// ---- Library/10_Machine/18_HMI_Handshake/DUTs/IOMonitor/ST_Wheelhouse_Layer.TcDUT
TYPE ST_Wheelhouse_Layer :
STRUCT
	Line : ARRAY[1..20] OF BOOL;
END_STRUCT
END_TYPE

// ---- Library/10_Machine/18_HMI_Handshake/DUTs/IOMonitor/UNI_HMI_WheelHouseInput.TcDUT
TYPE UNI_HMI_WheelHouseInput :
UNION
	arWheelHouseInput : ARRAY[1..400] OF BOOL;
	List :ST_WheelhouseInput;
END_UNION
END_TYPE

// ---- Library/10_Machine/18_HMI_Handshake/DUTs/IOMonitor/UNI_HMI_WheelHouseInput2.TcDUT
TYPE UNI_HMI_WheelHouseInput2 :
UNION
	arWheelHouseInput : ARRAY[1..400] OF BOOL;
	List :ST_WheelhouseInput;
END_UNION
END_TYPE

// ---- Library/10_Machine/18_HMI_Handshake/DUTs/Shipping/ST_Auto_Shipping.TcDUT
TYPE
    ST_Auto_Shipping :
    STRUCT
    END_STRUCT
END_TYPE

// ---- Library/10_Machine/18_HMI_Handshake/DUTs/Shipping/ST_HalfAuto_Shipping.TcDUT
TYPE
    ST_HalfAuto_Shipping :
    STRUCT
    END_STRUCT
END_TYPE

// ---- Library/10_Machine/18_HMI_Handshake/DUTs/Shipping/ST_HMI_ShippingArea.TcDUT
TYPE
    ST_HMI_ShippingArea :
    STRUCT
        //提供新的馬達
    END_STRUCT
END_TYPE

// ---- Library/10_Machine/18_HMI_Handshake/DUTs/Shipping/ST_Manual_Shipping.TcDUT
TYPE
    ST_Manual_Shipping :
    STRUCT
		FanucRobot : ST_Manual_FanucRobot;
    END_STRUCT
END_TYPE

// ---- Library/10_Machine/18_HMI_Handshake/DUTs/Status/ST_AllocateStatus.TcDUT
TYPE
    ST_AllocateStatus :
    STRUCT
    END_STRUCT
END_TYPE

// ---- Library/10_Machine/18_HMI_Handshake/DUTs/Status/ST_Auto_Status.TcDUT
TYPE ST_Auto_Status :
STRUCT
END_STRUCT
END_TYPE

// ---- Library/10_Machine/18_HMI_Handshake/DUTs/Status/ST_AXES_STATUS.TcDUT
TYPE ST_AXES_STATUS :
    STRUCT
        TurnTable       : ST_SINGLEAXIS_STATUS; 		// 圓盤 狀態
        Allocate        : ST_SINGLEAXIS_STATUS; 		// 圓帶 狀態
        Needle_X        : ST_SINGLEAXIS_STATUS; 		// 配針 X 狀態
        Needle_Y        : ST_SINGLEAXIS_STATUS; 		// 配針 Y 狀態
        OutRobot_X      : ST_SINGLEAXIS_STATUS; 		// 出料手臂 X 狀態
        OutRobot_Y      : ST_SINGLEAXIS_STATUS; 		// 出料手臂 Y 狀態
		RackMotor 		: ST_SINGLEAXIS_STATUS; 		// 補貨料架馬達 狀態
		ElvaterAxis		: ST_SINGLEAXIS_STATUS;			// 電梯 狀態
		HookAxis		: ST_SINGLEAXIS_STATUS;			// 勾盤 狀態
		FinishAxis		: ST_SINGLEAXIS_STATUS;			// 出料層架 狀態
    END_STRUCT
END_TYPE

// ---- Library/10_Machine/18_HMI_Handshake/DUTs/Status/ST_MotorStatus.TcDUT
TYPE
    ST_MotorStatus :
    STRUCT
        WareHouseCV_10          : ST_MotorMonitor;
        WareHouseCV_09          : ST_MotorMonitor;
        WareHouseCV_08          : ST_MotorMonitor;
        WareHouseCV_07          : ST_MotorMonitor;
        WareHouseCV_06          : ST_MotorMonitor;
        WareHouseCV_05          : ST_MotorMonitor;
        WareHouseCV_04          : ST_MotorMonitor;
        WareHouseCV_03          : ST_MotorMonitor;
        WareHouseCV_02          : ST_MotorMonitor;
        WareHouseCV_01          : ST_MotorMonitor;
        WareHouseCV_20          : ST_MotorMonitor;
        WareHouseCV_19          : ST_MotorMonitor;
        WareHouseCV_18          : ST_MotorMonitor;
        WareHouseCV_17          : ST_MotorMonitor;
        WareHouseCV_16          : ST_MotorMonitor;
        WareHouseCV_15          : ST_MotorMonitor;
        WareHouseCV_14          : ST_MotorMonitor;
        WareHouseCV_13          : ST_MotorMonitor;
        WareHouseCV_12          : ST_MotorMonitor;
        WareHouseCV_11          : ST_MotorMonitor;
        UpCV                    : ST_MotorMonitor;
        LowCV                   : ST_MotorMonitor;
        PullOutCV_A             : ST_MotorMonitor;
        PullOutCV_B             : ST_MotorMonitor;
        TransmitSameSideCV      : ST_MotorMonitor;
        TransmitDifferentSideCV : ST_MotorMonitor;
    END_STRUCT
END_TYPE

// ---- Library/10_Machine/18_HMI_Handshake/DUTs/Status/ST_SINGLEAXIS_STATUS.TcDUT
TYPE ST_SINGLEAXIS_STATUS :
    STRUCT
        ActPos    : LREAL; // Axis actual position with gear ratio
        ActVel    : LREAL; // Axis actual velocity with gear ratio
        MotorTemp : LREAL; // Motor current tempture, if motor doesn't have temp sensor, this value will be zero.
        DriveTemp : LREAL; // Driver current tempture
        Homed     : BOOL; // Axis has homed 
        Error     : BOOL; // Axis has error
        CmdDone   : BOOL; // Axis Cmd completed
    END_STRUCT
END_TYPE

// ---- Library/10_Machine/18_HMI_Handshake/DUTs/Status/ST_CylinderStatus.TcDUT
TYPE
    ST_CylinderStatus :
    STRUCT
        UpCV_FeedInPress1             : ST_CylinderMonitor;
        UpCV_FeedInPress2             : ST_CylinderMonitor;
        UpCV_DiameterPress            : ST_CylinderMonitor;
        UpCV_CamaraPress1             : ST_CylinderMonitor;
        UpCV_CamaraPress2             : ST_CylinderMonitor;
        UpCV_CamaraPress3             : ST_CylinderMonitor;
        UpCV_CamaraPress4             : ST_CylinderMonitor;
        UpCV_Block1                   : ST_CylinderMonitor;
        UpCV_Block2                   : ST_CylinderMonitor;
        UpCV_Block3                   : ST_CylinderMonitor;
        UpCV_DiameterHoriz            : ST_CylinderMonitor;
        UpCV_DiameterVert             : ST_CylinderMonitor;
        UpCV_DiameterClamp            : ST_CylinderMonitor;
        StackPush                     : ST_CylinderMonitor;
        PullOutCV_AsidePress1         : ST_CylinderMonitor;
        PullOutCV_AsidePress2         : ST_CylinderMonitor;
        PullOutCV_AsideBlock          : ST_CylinderMonitor;
        PullOutCV_BsidePress1         : ST_CylinderMonitor;
        PullOutCV_BsidePress2         : ST_CylinderMonitor;
        PullOutCV_BsideBlock          : ST_CylinderMonitor;
        LowCV_Press1                  : ST_CylinderMonitor;
        LowCV_Press2                  : ST_CylinderMonitor;
        LowCV_Press3                  : ST_CylinderMonitor;
        LowCV_Press4                  : ST_CylinderMonitor;
        LowCV_Block1                  : ST_CylinderMonitor;
        LowCV_Block2                  : ST_CylinderMonitor;
        AllocateRobot_LeftVert1       : ST_CylinderMonitor;
        AllocateRobot_LeftVert2       : ST_CylinderMonitor;
        AllocateRobot_RightVert1      : ST_CylinderMonitor;
        AllocateRobot_RightVert2      : ST_CylinderMonitor;
        AllocateRobot_LeftClamp1      : ST_CylinderMonitor;
        AllocateRobot_LeftClamp2      : ST_CylinderMonitor;
        AllocateRobot_RightClamp1     : ST_CylinderMonitor;
        AllocateRobot_RightClamp2     : ST_CylinderMonitor;
        RoundBelt_WorkZone_Press      : ST_CylinderMonitor;
        RoundBelt_WorkZone_Plug       : ST_CylinderMonitor;
        RoundBelt_ChargeZone_Plug     : ST_CylinderMonitor;
        RoundBelt_TransmitCVZone_Plug : ST_CylinderMonitor;
        OutRobot_AsideVert            : ST_CylinderMonitor;
        OutRobot_BsideVert            : ST_CylinderMonitor;
        OutRobot_AsideClamp           : ST_CylinderMonitor;
        OutRobot_BsideClamp           : ST_CylinderMonitor;
        TransmitCV_CamaraHoriz        : ST_CylinderMonitor;
        DifferentSizeCV_Press2        : ST_CylinderMonitor;
        DifferentSizeCV_Press1        : ST_CylinderMonitor;
        DifferentSizeCV_Block1        : ST_CylinderMonitor;
        SameSizeCV_Press4             : ST_CylinderMonitor;
        SameSizeCV_Press3             : ST_CylinderMonitor;
        SameSizeCV_Press2             : ST_CylinderMonitor;
        SameSizeCV_Press1             : ST_CylinderMonitor;
        SameSizeCV_Block2             : ST_CylinderMonitor;
        SameSizeCV_Block1             : ST_CylinderMonitor;
        Turntable_Press               : ST_CylinderMonitor;
    END_STRUCT
END_TYPE

// ---- Library/10_Machine/18_HMI_Handshake/DUTs/Status/ST_HalfAuto_Status.TcDUT
TYPE ST_HalfAuto_Status :
STRUCT
END_STRUCT
END_TYPE

// ---- Library/10_Machine/18_HMI_Handshake/DUTs/Status/ST_HMI_MachineStatus.TcDUT
TYPE
    ST_HMI_MachineStatus :
    STRUCT
        Axes      : ST_AXES_STATUS;	  //馬達狀態
        Cylinders : ST_CylinderStatus;//汽缸狀態
        Motor     : ST_MotorStatus;	  //軌道狀態
    END_STRUCT
END_TYPE

// ---- Library/10_Machine/18_HMI_Handshake/DUTs/Status/ST_Manual_Status.TcDUT
TYPE ST_Manual_Status :
STRUCT
	Cylinders : ST_CylinderStatus;
END_STRUCT
END_TYPE

// ---- Library/10_Machine/18_HMI_Handshake/DUTs/Status/ST_ShippingStatus.TcDUT
TYPE ST_ShippingStatus :
STRUCT
END_STRUCT
END_TYPE

// ---- Library/10_Machine/18_HMI_Handshake/DUTs/Status/ST_StorageStatus.TcDUT
TYPE ST_StorageStatus :
STRUCT
END_STRUCT
END_TYPE

// ---- Library/10_Machine/18_HMI_Handshake/DUTs/Storage/ST_Auto_Storage.TcDUT
TYPE
    ST_Auto_Storage :
    STRUCT
    END_STRUCT
END_TYPE

// ---- Library/10_Machine/18_HMI_Handshake/DUTs/Storage/ST_HalfAuto_Storage.TcDUT
TYPE
    ST_HalfAuto_Storage :
    STRUCT
    END_STRUCT
END_TYPE

// ---- Library/10_Machine/18_HMI_Handshake/DUTs/Storage/ST_HMI_ControlConvery.TcDUT
TYPE
    ST_HMI_ControlConvery :
    STRUCT
		//A倉軌道
        WareHouseCV_10  : ST_MotorCommand;
        WareHouseCV_09  : ST_MotorCommand;
        WareHouseCV_08  : ST_MotorCommand;
        WareHouseCV_07  : ST_MotorCommand;
        WareHouseCV_06  : ST_MotorCommand;
        WareHouseCV_05  : ST_MotorCommand;
        WareHouseCV_04  : ST_MotorCommand;
        WareHouseCV_03  : ST_MotorCommand;
        WareHouseCV_02  : ST_MotorCommand;
        WareHouseCV_01  : ST_MotorCommand;
		//B倉軌道
        WareHouseCV_20  : ST_MotorCommand;
        WareHouseCV_19  : ST_MotorCommand;
        WareHouseCV_18  : ST_MotorCommand;
        WareHouseCV_17  : ST_MotorCommand;
        WareHouseCV_16  : ST_MotorCommand;
        WareHouseCV_15  : ST_MotorCommand;
        WareHouseCV_14  : ST_MotorCommand;
        WareHouseCV_13  : ST_MotorCommand;
        WareHouseCV_12  : ST_MotorCommand;
        WareHouseCV_11  : ST_MotorCommand;
		
        UpCV            : ST_Manual_UpCV;			//上層入料軌道
        LowCV        	: ST_Manual_LowCV;			//下層出料軌道
		PullOutCV       : ST_Manual_PullOutCV;      // 空盒以及拔針軌道
        TransCV         : ST_Manual_TransCV;        // 同尺寸以及配針軌道
    END_STRUCT
END_TYPE

// ---- Library/10_Machine/18_HMI_Handshake/DUTs/Storage/ST_Manual_FanucRobot.TcDUT
TYPE ST_Manual_FanucRobot :
STRUCT
	ClampA_Open  		: BOOL; // True: set clampA open 
	ClampA_Close 		: BOOL; // True: Set ClampA Close
	ClampB_Open  		: BOOL; // True: Set ClampB Open
	ClampB_Close 		: BOOL; // True: Set ClampB Close
	ByPassClampSensor   : BOOL; // True : Bypass clampA and clampB
END_STRUCT
END_TYPE

// ---- Library/10_Machine/18_HMI_Handshake/DUTs/Storage/ST_Manual_Rack.TcDUT
TYPE ST_Manual_Rack :
STRUCT
	Axis                : ST_Manual_Axis; // RoundBelt Axis controll
END_STRUCT
END_TYPE

// ---- Library/10_Machine/18_HMI_Handshake/DUTs/Storage/ST_Manual_UpCV.TcDUT
TYPE
    ST_Manual_UpCV :
    STRUCT
        FeedInPress1  : ST_SignleValve;
        FeedInPress2  : ST_SignleValve;
        DiameterPress : ST_SignleValve;
        CamaraPress1  : ST_SignleValve;
        CamaraPress2  : ST_SignleValve;
        CamaraPress3  : ST_SignleValve;
        CamaraPress4  : ST_SignleValve;
        Block1        : ST_SignleValve;
        Block2        : ST_SignleValve;
        Block3        : ST_SignleValve;
        DiameterHoriz : ST_SignleValve;
        DiameterVert  : ST_SignleValve;
        DiameterClamp : ST_SignleValve;
        StackPush     : ST_SignleValve;
		CameraBlow	  : BOOL;
        UpCV          : ST_MotorCommand;
    END_STRUCT
END_TYPE

// ---- Library/10_Machine/18_HMI_Handshake/DUTs/Storage/ST_Manual_LowCV.TcDUT
TYPE
    ST_Manual_LowCV :
    STRUCT
        Press1 : ST_SignleValve;
        Press2 : ST_SignleValve;
        Press3 : ST_SignleValve;
        Press4 : ST_SignleValve;
        Block1 : ST_SignleValve;
        Block2 : ST_SignleValve;
        LowCV  : ST_MotorCommand;
    END_STRUCT
END_TYPE

// ---- Library/10_Machine/18_HMI_Handshake/DUTs/Storage/ST_Manual_Storage.TcDUT
TYPE
    ST_Manual_Storage :
    STRUCT
        WareHouseCV_10 : ST_MotorCommand;
        WareHouseCV_09 : ST_MotorCommand;
        WareHouseCV_08 : ST_MotorCommand;
        WareHouseCV_07 : ST_MotorCommand;
        WareHouseCV_06 : ST_MotorCommand;
        WareHouseCV_05 : ST_MotorCommand;
        WareHouseCV_04 : ST_MotorCommand;
        WareHouseCV_03 : ST_MotorCommand;
        WareHouseCV_02 : ST_MotorCommand;
        WareHouseCV_01 : ST_MotorCommand;
        WareHouseCV_20 : ST_MotorCommand;
        WareHouseCV_19 : ST_MotorCommand;
        WareHouseCV_18 : ST_MotorCommand;
        WareHouseCV_17 : ST_MotorCommand;
        WareHouseCV_16 : ST_MotorCommand;
        WareHouseCV_15 : ST_MotorCommand;
        WareHouseCV_14 : ST_MotorCommand;
        WareHouseCV_13 : ST_MotorCommand;
        WareHouseCV_12 : ST_MotorCommand;
        WareHouseCV_11 : ST_MotorCommand;
        UpCV           : ST_Manual_UpCV;
        LowCV          : ST_Manual_LowCV;
		FanucRobot : ST_Manual_FanucRobot;
		RackMotor :ST_Manual_Rack;
    END_STRUCT
END_TYPE

// ---- Library/10_Machine/18_HMI_Handshake/OLD_DUTs/DataCore/E_BoxHookPoint.TcDUT
{attribute 'qualified_only'}
{attribute 'strict'}
TYPE E_BoxHookPoint :
(
	
	Origin 		:= 0,
	Station_1	:= 1,
	Station_2	:= 2,
	Station_3	:= 3,
	Station_4	:= 4,
	Station_5	:= 5,
	Station_6	:= 6,
	Station_7	:= 7,
	Station_8	:= 8,
	Station_9	:= 9,
	
);
END_TYPE

// ---- Library/10_Machine/18_HMI_Handshake/OLD_DUTs/DataCore/E_BufferArea.TcDUT
{attribute 'qualified_only'}
{attribute 'strict'}
TYPE E_BufferArea :
(
	enum_member 	:= 0,
	buffers_1		:= 1,
	buffers_2		:= 2,
	buffers_3		:= 3,
	buffers_4		:= 4,
	buffers_5		:= 5,
	buffers_6		:= 6,
	buffers_7		:= 7,
	buffers_8		:= 8,
	buffers_9		:= 9,
	buffers_10		:= 10,
	buffers_11		:= 11,
	buffers_12		:= 12,
	buffers_13		:= 13,
	buffers_14		:= 14,
	buffers_15		:= 15,
	buffers_16		:= 16,
	buffers_17		:= 17,
	buffers_18		:= 18,
	buffers_19		:= 19,
	buffers_20		:= 20,
	buffers_21		:= 21,
	buffers_22		:= 22,
	buffers_23		:= 23,
	buffers_24		:= 24,
	buffers_25		:= 25,
	buffers_26		:= 26,
	buffers_27		:= 27,
	buffers_28		:= 28,
	buffers_29		:= 29,
	buffers_30		:= 30,
	buffers_31		:= 31,
	buffers_32		:= 32,
	buffers_33		:= 33,
	buffers_34		:= 34,
	buffers_35		:= 35,
	buffers_36		:= 36,
	buffers_37		:= 37,
	buffers_38		:= 38,
	buffers_39		:= 39,
	buffers_40		:= 40,
);
END_TYPE

// ---- Library/10_Machine/18_HMI_Handshake/OLD_DUTs/DataCore/E_BoxStatus.TcDUT
{attribute 'qualified_only'}
{attribute 'strict'}
TYPE E_BoxStatus :
(
	EmptyBox 			:= 0,
	FullBox  			:= 1,
	NeedleBox			:= 2,
	NeedleRemoveBox		:= 3,
);
END_TYPE

// ---- Library/10_Machine/18_HMI_Handshake/OLD_DUTs/DataCore/E_LayerPoint.TcDUT
{attribute 'qualified_only'}
{attribute 'strict'}
TYPE E_LayerPoint :
(
	Origin 		:= 0,
	Station_1	:= 1,
	Station_2	:= 2,
	Station_3	:= 3,
	Station_4	:= 4,
	Station_5	:= 5,
	Station_6	:= 6,
);
END_TYPE

// ---- Library/10_Machine/18_HMI_Handshake/OLD_DUTs/DataCore/E_MachineMode.TcDUT
{attribute 'qualified_only'}
{attribute 'strict'}
TYPE E_MachineMode :
(
	UNDEFINE := 0,
	MANUAL	:=1		  ,
	AUTO	:=2		  ,
	SERVICE :=3,
	ModeSelect:=99
);
END_TYPE

// ---- Library/10_Machine/18_HMI_Handshake/OLD_DUTs/DataCore/E_mode.TcDUT
{attribute 'qualified_only'}
{attribute 'strict'}
TYPE E_mode :
(
	default 	:= 0,
	fullmode 	:= 1,
	even 		:= 2,
	odd 		:= 3,
);
END_TYPE

// ---- Library/10_Machine/18_HMI_Handshake/OLD_DUTs/DataCore/E_NeedleClip.TcDUT
{attribute 'qualified_only'}
{attribute 'strict'}
TYPE E_NeedleClip :
(
	clip_A		:= 0,
	clip_B		:= 1,
	clip_C		:= 2,
	clip_D		:= 3,
);
END_TYPE

// ---- Library/10_Machine/18_HMI_Handshake/OLD_DUTs/DataCore/E_Location.TcDUT
{attribute 'qualified_only'}
{attribute 'strict'}
TYPE E_Location :
(
	default				:= 0,	//不作動
	UpConvery			:= 1,	//入料上層軌道
	LowConvery			:= 2,	//出料下層軌道
	OutPullconveryLeft 	:= 3,	//待研磨軌道
	OutPullconveryRight := 4,	//取空盒軌道
	Warehouse 			:= 5,	//倉儲
	Buffers				:= 6,   //緩衝區
	SameConvery			:= 7, 	//同尺寸軌道
	DifferentConvery	:= 8,	//不同尺寸軌道
	AllocateLeft		:= 9,	//圓帶左盒
	AllocatrRight		:= 10,	//圓帶右盒
)UINT;
END_TYPE

// ---- Library/10_Machine/18_HMI_Handshake/OLD_DUTs/DataCore/E_MachineTask.TcDUT
{attribute 'qualified_only'}
{attribute 'strict'}
TYPE E_MachineTask :
(
	//當前機台任務狀態
	default						:= 0,//尚未有任務
	Feeding						:= 1,//入料
	Discharge					:= 2,//出料
	Needle						:= 3,//配針啟動
	NeedleRemove				:= 4,//拔針啟動
	NeedleAllocate				:= 5,//配針領料
	NeedleRemoveAllocate		:= 6,//拔針領料
	WarehouseBack 				:= 7,//配針回倉
	WarehouseBackRemove 		:= 8,//拔針回倉
	SheepingPicture				:= 9,//出料拍照
	NeedleRemovePicture			:= 10,//拔針拍照
	NeedleChangeBox				:= 11,//配針換盒
	NeedleRemoveChangeBox		:= 12,//拔針換盒
	NeedleChangeAllocate		:= 13,//配針換圓帶
	NeedleRemoveChangeAllocate	:= 14,//拔針換圓帶 
	SixRobotWarehouseAction 	:= 15,//手臂倉儲動作
	SixRobotBuffersAction		:= 16,//手臂緩衝區動作
	TaskDone					:= 17,//任務完成
	Alarm 						:= 18,//錯誤發生
);
END_TYPE

// ---- Library/10_Machine/18_HMI_Handshake/OLD_DUTs/DataCore/E_NeedlePoint.TcDUT
TYPE E_NeedlePoint :
STRUCT
	default				:0,
	AllocateLeft 		:1,
	AllocateRight 		:2,
	TurntableLeft       :3,
	TurntableRight		:4,
END_STRUCT
END_TYPE

// ---- Library/10_Machine/18_HMI_Handshake/OLD_DUTs/DataCore/E_OutRobotClip.TcDUT
{attribute 'qualified_only'}
{attribute 'strict'}
TYPE E_OutRobotClip :
(
	clip_A		:= 0,
	clip_B		:= 1,
);
END_TYPE

// ---- Library/10_Machine/18_HMI_Handshake/OLD_DUTs/DataCore/E_OutRobotPoint.TcDUT
{attribute 'qualified_only'}
{attribute 'strict'}
TYPE E_OutRobotPoint :
(
	default 			:= 0,
	SameConvery 		:= 1,
	DifferentConvery	:= 2,
	TurnTableLeft		:= 3,
	TurnTableRight		:= 3,

	
);
END_TYPE

// ---- Library/10_Machine/18_HMI_Handshake/OLD_DUTs/DataCore/E_PlateHookPoint.TcDUT
{attribute 'qualified_only'}
{attribute 'strict'}
TYPE E_PlateHookPoint :
(
	Origin 		:= 0,
	Station_1	:= 1,
	Station_2	:= 2,
	Station_3	:= 3,
	Station_4	:= 4,
	Station_5	:= 5,
	Station_6	:= 6,
	Station_7	:= 7,
	Station_8	:= 8,
	Station_9	:= 9,
);
END_TYPE

// ---- Library/10_Machine/18_HMI_Handshake/OLD_DUTs/DataCore/st_AllocatingNeedleInfo.TcDUT
TYPE st_AllocatingNeedleInfo :
STRUCT
	NeedleLocation		: INT;	//針位，0~49
	Box					: UINT;	//盒位，0~3
	Clip				: INT;	//使用夾爪，0~3(可新增到5)
	Station				: UINT;	//圓帶站點 ，(放針時無效) 0..39
	CycleStart			: BOOL;	//取到此針後執行放針，討論放針做為作動依據
END_STRUCT
END_TYPE

// ---- Library/10_Machine/18_HMI_Handshake/OLD_DUTs/DataCore/ST_AllocationJobBatchModeInfo.TcDUT
TYPE ST_AllocationJobBatchModeInfo :
STRUCT
	PickingNeedleInfo			: ARRAY[0..3] OF st_AllocatingNeedleInfo;	//取針資料
	PlacingNeedleInfo			: ARRAY[0..3] OF st_AllocatingNeedleInfo;	//放針資料
	FastMode					: BOOL;
	SyncMode					: BOOL;
	ID							: INT;   // -1 means null , do not use
END_STRUCT
END_TYPE

// ---- Library/10_Machine/18_HMI_Handshake/OLD_DUTs/DataCore/st_BoxHookStationMove.TcDUT
TYPE st_BoxHookStationMove :
STRUCT
	BoxHookPoint	: E_BoxHookPoint;
	Handshake		: ST_HandshakeBase;
END_STRUCT
END_TYPE

// ---- Library/10_Machine/18_HMI_Handshake/OLD_DUTs/DataCore/ST9_ChangeBox.TcDUT
TYPE ST9_ChangeBox :
STRUCT
	Info 			: ST1_ChangeBoxInfo;
	Handshake		: ST_HandshakeBase;
END_STRUCT
END_TYPE

// ---- Library/10_Machine/18_HMI_Handshake/OLD_DUTs/DataCore/st_ChangeBoxesData.TcDUT
TYPE st_ChangeBoxesData :
STRUCT
	//圓帶位置
	AllocationNo			: E_StationOrder;//1~40 
	//倉儲位置
	StorageInfor			: INT; //1~400
	//盒子順序
	BoxOrder				: INT;//1~10
	//數量
	Num						: INT;//1~50
END_STRUCT
END_TYPE

// ---- Library/10_Machine/18_HMI_Handshake/OLD_DUTs/DataCore/ST0_ChangeBoxesInfo.TcDUT
TYPE ST0_ChangeBoxesInfo :
STRUCT
	ChangeBoxesData 	:ARRAY[0..40] OF st_ChangeBoxesData;
END_STRUCT
END_TYPE

// ---- Library/10_Machine/18_HMI_Handshake/OLD_DUTs/DataCore/ST1_ChangeBoxInfo.TcDUT
TYPE ST1_ChangeBoxInfo :
STRUCT
	CheckedChangeBox		:	BOOL;
	ChangeBox 				:	ST0_ChangeBoxesInfo;
	HandShake				:  	st_HandshakeBase;
END_STRUCT
END_TYPE

// ---- Library/10_Machine/18_HMI_Handshake/OLD_DUTs/DataCore/st_LayerStationMove.TcDUT
TYPE st_LayerStationMove :
STRUCT
	LayerPoint		: E_LayerPoint;
	Handshake		: ST_HandshakeBase;
END_STRUCT
END_TYPE

// ---- Library/10_Machine/18_HMI_Handshake/OLD_DUTs/DataCore/ST_Mode.TcDUT
TYPE ST_Mode :
STRUCT
	TargetMode	:E_MachineMode := E_MachineMode.UNDEFINE; 	
	CurrentMode :E_MachineMode:=E_MachineMode.ModeSelect;
	HandshakeBase : st_HandshakeBase;
END_STRUCT
END_TYPE

// ---- Library/10_Machine/18_HMI_Handshake/OLD_DUTs/DataCore/ST_Output.TcDUT
TYPE ST_Output :
STRUCT
		Info						: ARRAY[0..300] OF ST_DischargeDataInfo;
		HandShake					: ST_HandshakeBase;
END_STRUCT
END_TYPE

// ---- Library/10_Machine/18_HMI_Handshake/OLD_DUTs/DataCore/ST_DischargeDataInfo.TcDUT
TYPE ST_DischargeDataInfo :
STRUCT
	//倉儲儲位
	StorageInfor	:INT;
	//盒子順序
	BoxOrder 		:INT;
	//放置位置
	PutPlace 		:E_Location;
END_STRUCT
END_TYPE

// ---- Library/10_Machine/18_HMI_Handshake/OLD_DUTs/DataCore/ST_Feeding.TcDUT
TYPE ST_Feeding :
STRUCT
		Info		: ST_FeedingDataInfo;
		Feeback		: ST_FeedingDataFeeback;
		Handshake	: ST_HandshakeBase;
END_STRUCT
END_TYPE

// ---- Library/10_Machine/18_HMI_Handshake/OLD_DUTs/DataCore/ST_FeedingDataFeeback.TcDUT
TYPE ST_FeedingDataFeeback :
STRUCT
	Camera 					:BOOL;
	CameraDiameter 			:BOOL;
	
END_STRUCT
END_TYPE

// ---- Library/10_Machine/18_HMI_Handshake/OLD_DUTs/DataCore/ST_FeedingDataInfo.TcDUT
TYPE ST_FeedingDataInfo :
STRUCT
	BoxCameraDone 					: BOOL;//拍照結束
	CameraDiameterRequest 			: BOOL;//外徑需求
	CameraDiameterDone 				: BOOL;//外徑拍照結束
	FirstBoxLocation 				: E_Location;//第一盒位置
	SecondBoxLocation 				: E_Location;//第二盒位置
	FirstBoxStorageInfor			:INT;//第一盒到倉儲的位置
	SecondBoxStorageInfor			:INT;//第二盒到倉儲的位置
	stopFeeding						:BOOL;//中斷入料
END_STRUCT
END_TYPE

// ---- Library/10_Machine/18_HMI_Handshake/OLD_DUTs/DataCore/ST_GetBox.TcDUT
TYPE ST_GetBox :
STRUCT
	Info 			: ARRAY[0..200] OF ST_GetBoxInfo;
	//盒數
	NeedBox			:INT;
	//資料交握確認
	HandShake		: st_HandshakeBase;
END_STRUCT
END_TYPE

// ---- Library/10_Machine/18_HMI_Handshake/OLD_DUTs/DataCore/st_NeedleAction.TcDUT
TYPE st_NeedleAction :
STRUCT
	Clip				: E_NeedleClip;
	NeedlePoint			: E_NeedlePoint;
	Handshake			: ST_HandshakeBase;
END_STRUCT
END_TYPE

// ---- Library/10_Machine/18_HMI_Handshake/OLD_DUTs/DataCore/st_NeedleActionBatch.TcDUT
TYPE st_NeedleActionBatch :
STRUCT
	mode			: E_mode;
	Handshake		: ST_HandshakeBase;
END_STRUCT
END_TYPE

// ---- Library/10_Machine/18_HMI_Handshake/OLD_DUTs/DataCore/ST_NeedleAllocatefeeback.TcDUT
TYPE ST_NeedleAllocatefeeback :
STRUCT
	//領取盒子的狀態
	BoxStatus		:		E_BoxStatus;
	//所需盒數
	Box				:       INT;
END_STRUCT
END_TYPE

// ---- Library/10_Machine/18_HMI_Handshake/OLD_DUTs/DataCore/ST_NeedleAllocateinfo.TcDUT
TYPE ST_NeedleAllocateinfo :
STRUCT
		//告知位置
		WarehouseGetBox		: ARRAY[0..300] OF ST_WarehouseGetBox;
END_STRUCT
END_TYPE

// ---- Library/10_Machine/18_HMI_Handshake/OLD_DUTs/DataCore/ST_ChangeAllocate.TcDUT
TYPE ST_ChangeAllocate :
STRUCT
		Info 						: ST_NeedleChangeAllocateInfo;
		Handshake					: ST_HandshakeBase;
END_STRUCT
END_TYPE

// ---- Library/10_Machine/18_HMI_Handshake/OLD_DUTs/DataCore/ST_NeedleChangeAllocateInfo.TcDUT
TYPE ST_NeedleChangeAllocateInfo :
STRUCT
	//確認是否要換
	CheckedChangeAllocate	:  BOOL;
	ChangeAllocate 			:  ARRAY[0..40] OF st_AllocationData;
END_STRUCT
END_TYPE

// ---- Library/10_Machine/18_HMI_Handshake/OLD_DUTs/DataCore/ST_NeedleRemove.TcDUT
TYPE ST_NeedleRemove :
STRUCT
	//配針動作資料
		NeedleInfo					: ARRAY[0..2000] OF ST_AllocationJobBatchModeInfo; 
	//初始圓帶資料
		AllocationInfoData			: ARRAY[0..40] OF st_AllocationData;
	//拔針盒數
		NeedleRemoveCount			:INT;
	//資料交握確認
		HandShake					: st_HandshakeBase;
END_STRUCT
END_TYPE

// ---- Library/10_Machine/18_HMI_Handshake/OLD_DUTs/DataCore/ST_NeedleRemoveAllocate.TcDUT
TYPE ST_NeedleRemoveAllocate :
STRUCT
	Info 	: ST_NeedleAllocateinfo;
END_STRUCT
END_TYPE

// ---- Library/10_Machine/18_HMI_Handshake/OLD_DUTs/DataCore/st_OutRobotMove.TcDUT
TYPE st_OutRobotMove :
STRUCT
	Clip				: E_OutRobotClip;
	OutRobotPoint		: E_OutRobotPoint;
	Handshake			: ST_HandshakeBase;
END_STRUCT
END_TYPE

// ---- Library/10_Machine/18_HMI_Handshake/OLD_DUTs/DataCore/ST_PCTask.TcDUT
TYPE ST_PCTask :
STRUCT
	Needle			:BOOL;//配針
	NeedleRemove	:BOOL;//拔針
	Feeding			:BOOL;//入料
	Output			:BOOL;//出料
END_STRUCT
END_TYPE

// ---- Library/10_Machine/18_HMI_Handshake/OLD_DUTs/DataCore/st_PlateHookStationMove.TcDUT
TYPE st_PlateHookStationMove :
STRUCT
	PlateHookPoint		: E_PlateHookPoint;
	Handshake			: ST_HandshakeBase;
END_STRUCT
END_TYPE

// ---- Library/10_Machine/18_HMI_Handshake/OLD_DUTs/DataCore/ST_PlateOrder.TcDUT
TYPE ST_PlateOrder :
STRUCT
	PlateOrder:INT;
	BoxStatus:E_BoxStatus;
END_STRUCT
END_TYPE

// ---- Library/10_Machine/18_HMI_Handshake/OLD_DUTs/DataCore/E_StationOrder.TcDUT
{attribute 'qualified_only'}
{attribute 'strict'}
TYPE E_StationOrder :
(
	enum_member := 0,
	station_1	:= 1,
	station_2	:= 2,
	station_3	:= 3,
	station_4	:= 4,
	station_5	:= 5,
	station_6	:= 6,
	station_7	:= 7,
	station_8	:= 8,
	station_9	:= 9,
	station_10	:= 10,
	station_11	:= 11,
	station_12	:= 12,
	station_13	:= 13,
	station_14	:= 14,
	station_15	:= 15,
	station_16	:= 16,
	station_17	:= 17,
	station_18	:= 18,
	station_19	:= 19,
	station_20	:= 20,
	station_21	:= 21,
	station_22	:= 22,
	station_23	:= 23,
	station_24	:= 24,
	station_25	:= 25,
	station_26	:= 26,
	station_27	:= 27,
	station_28	:= 28,
	station_29	:= 29,
	station_30	:= 30,
	station_31	:= 31,
	station_32	:= 32,
	station_33	:= 33,
	station_34	:= 34,
	station_35	:= 35,
	station_36	:= 36,
	station_37  := 37;
	station_38	:= 38,
	station_39	:= 39,
	station_40	:= 40,
);
END_TYPE

// ---- Library/10_Machine/18_HMI_Handshake/OLD_DUTs/DataCore/ST_ACTIVEDATA.TcDUT
TYPE ST_ACTIVEDATA :
STRUCT
	//當前任務狀態
	MachineTask					: E_MachineTask
	//配針換盒
	RotateChangeBoxData 		: ST_RotateChangeBoxData;
	//拔針換盒
	RotateChangeRemoveBoxData 	: ST_RotateChangeBoxData;
	//切換圓帶
	RotateChangeData 			: ST_RotateChangeData;
	//手臂出倉完成
	SixRobotGet 				: ST_SixRobotGet;
	//手臂入倉完成
	SixRobotPut 				: ST_SixRobotGet;
	//領取盒滿
	GetFullBox					: ST_GetFullBox
	//領取待拔針
	GetRemoveBox 				: ST_GetRemoveBox
	//錯誤
	AutoMode_ErrorHandle 		: ST_Alarm;
END_STRUCT
END_TYPE

// ---- Library/10_Machine/18_HMI_Handshake/OLD_DUTs/DataCore/ST_ActiveResult.TcDUT
TYPE ST_ActiveResult :
STRUCT
	//錯誤
	AutoMode_ErrorHandle 		: ST_Alarm;
END_STRUCT
END_TYPE

// ---- Library/10_Machine/18_HMI_Handshake/OLD_DUTs/DataCore/ST_AllocationData.TcDUT
TYPE ST_AllocationData
STRUCT
	//圓帶位置 0代表沒有盒子
	AllocationNo			: E_StationOrder;//1~40 
	//倉儲位置
	StorageInfor			: INT; //1~400
	//倉儲盒子順序
	BoxOrder				: INT;//1~10
	//換盒次數
	ChangeBoxCount          : INT;
	//針數量
	
	//
	//SIZE  				:DOUBLE
	//
	//CYCLE					:INT
	
	Num						: INT;//1~50
END_STRUCT
END_TYPE

// ---- Library/10_Machine/18_HMI_Handshake/OLD_DUTs/DataCore/ST_AllocationInfo.TcDUT
TYPE ST_AllocationInfo:
STRUCT
		AllocationData 	:ARRAY[0..40] OF st_AllocationData;
END_STRUCT
END_TYPE

// ---- Library/10_Machine/18_HMI_Handshake/OLD_DUTs/DataCore/ST_AllocationJobBatchMode_Reverse.TcDUT
TYPE ST_AllocationatchMode_Reverse:
STRUCT
//配針動作資料
	NeedleInfo					: ARRAY[0..2000] OF ST_AllocationJobBatchModeInfo; 
//圓帶資料
	AllocationInfoData			: ARRAY[0..6] OF ST_AllocationInfo;
//資料交握確認
	HandShake					: st_HandshakeBase;
END_STRUCT
 END_TYPE

// ---- Library/10_Machine/18_HMI_Handshake/OLD_DUTs/DataCore/st_ADSBaseParaCore.TcDUT
TYPE st_ADSBaseParaCore :
	STRUCT
		//配針手臂在圓帶的盒的左右的間距
		Allocate_box_leftandRight_Distance: LREAL;
	    //配針手臂在圓帶的盒的上下的間距
		Allocate_box_UpandDown_Distance   : LREAL;
		//配針手臂在圓帶的盒的間距
		Allocate_Box_Between_BBox_Distance:LREAL;
		//配針手臂在圓盤盒的左右間距
		TurnTable_leftandRight_Distance: LREAL;
		//配針手臂在圓盤盒的上下的間距
		TurnTable_UpandDown_Distance: LREAL;
		//配針手臂在圓盤的盒的間距
		TurnTable_Box_Between_BBox_Distance:LREAL;
		//圓帶的初始位置[1]
		Allocate_Original_Position:LREAL;
		//圓盤初始位置[2]
		TurnTable_Original_Position:LREAL;
		//出料軸X初始位置[3]
		OutRobotX_Original_Position:LREAL;
		//出料軸Y初始位置[4]
		OutRobotY_Original_Position:LREAL;
		//出料軸R初始位置[5]
		OutRobotR_Original_Position:LREAL;
		//配針軸X初始位置[6]
		AllocateRobotX_Original_Position:LREAL;
		//配針軸Y初始位置[7]
		AllocateRobotY_Original_Position:LREAL;
		//電梯初始位置[8]
		ElvaterAxis_Original_Position:LREAL;
		//勾盤初始位置[9]
		HookAxis_Original_Position:LREAL;
		//成品區層架初始位置[10]
		FinishAxisUPDownAxis_Original_Position:LREAL;
		//分選區初始位置[11]
		WarehouseAxis_Original_Position:LREAL;
       //圓帶與圓帶的間距
		Allocate_Box_Box_Distance:LREAL;
		//出料區盒與盒間距
		OutBoxBoxDistance:LREAL;
		//背隙補償 for 圓帶
		lrRotateBacklash :LREAL;
		//移動
		BuzzTime		 :LREAL;
		//蜂鳴器持續時間 in second
  		Excute:BOOL;
   		 //完成
		Done:BOOL;
	
	END_STRUCT
END_TYPE

// ---- Library/10_Machine/18_HMI_Handshake/OLD_DUTs/DataCore/st_ADSMotoCore.TcDUT
//上位系統給控制器馬達參數結構
TYPE st_ADSMotoCore  :
STRUCT
	//馬達名稱
	MotoName:STRING;
	//是否使用軟體極限
	UseSoftlimit:BOOL;
	//軟體負極限
	SoftNegative:LREAL;
	//軟體正極限
	SoftPositive:LREAL;
	//速度
	VCC:LREAL;
	//加速
	ACC:LREAL;
	//減速
	DCC:LREAL;
	//Jerk
	Jerk:LREAL;
	//back home abs
	home_abs:LREAL;
	//執行
	Excute:BOOL;
	//馬達是否完成移動
	Done:BOOL;
	
END_STRUCT
END_TYPE

// ---- Library/10_Machine/18_HMI_Handshake/OLD_DUTs/DataCore/st_ADSMotoMoveCore.TcDUT
//上位系統給控制器馬達參數結構
TYPE st_ADSMotoMoveCore  :
STRUCT
	//馬達名稱
	MotoName:STRING;
	//是否使用軟體極限
  	AbsolutionPosition:LREAL;
	//執行
	Excute:BOOL;
	//馬達是否完成移動
	Done:BOOL;
	
	//home
	Home:BOOL;
	HomeDone:BOOL;
END_STRUCT
END_TYPE

// ---- Library/10_Machine/18_HMI_Handshake/OLD_DUTs/DataCore/st_AllocateParameterCore.TcDUT
//散配區座標結構
TYPE st_AllocateParameterCore  :
STRUCT
  	fName  :STRING;
 	index:  LREAL;
	X      :LREAL;
	Y      :LREAL;
	Clip   :LREAL;
	Excute:BOOL;
	Done  :BOOL;
END_STRUCT
END_TYPE

// ---- Library/10_Machine/18_HMI_Handshake/OLD_DUTs/DataCore/st_RegionHome.TcDUT
TYPE st_RegionHome :
STRUCT
	Homed	:BOOL;
	HandShake :st_HandshakeBase;
END_STRUCT
END_TYPE

// ---- Library/10_Machine/18_HMI_Handshake/OLD_DUTs/DataCore/ST_SheepingPicture.TcDUT
TYPE ST_SheepingPicture :
STRUCT
	Info 						: ST_SheepingPictureInfo;
	Feeback 					: ST_SheepingPictureFeeback;
	Handshake	: ST_HandshakeBase;
END_STRUCT
END_TYPE

// ---- Library/10_Machine/18_HMI_Handshake/OLD_DUTs/DataCore/ST_SheepingPictureFeeback.TcDUT
TYPE ST_SheepingPictureFeeback :
STRUCT
	CameraPositionDone : BOOL;
END_STRUCT
END_TYPE

// ---- Library/10_Machine/18_HMI_Handshake/OLD_DUTs/DataCore/ST_SheepingPictureInfo.TcDUT
TYPE ST_SheepingPictureInfo :
STRUCT
	CameraDone	:BOOL;
END_STRUCT
END_TYPE

// ---- Library/10_Machine/18_HMI_Handshake/OLD_DUTs/DataCore/ST_SixRobotAction.TcDUT
TYPE ST_SixRobotAction :
STRUCT
	Info		:ST_SixRobotActionInfo;
	Feeback		:ST_SixRobotActionFeeback;
	Handshake	: ST_HandshakeBase;
END_STRUCT
END_TYPE

// ---- Library/10_Machine/18_HMI_Handshake/OLD_DUTs/DataCore/ST_SixRobotActionFeeback.TcDUT
TYPE ST_SixRobotActionFeeback :
STRUCT
	SixRobotState			:E_MachineMode
	GET						:BOOL
	//倉儲位置
	A_StorageInfor			: INT; //1~400
	//倉儲位置
	B_StorageInfor			: INT; //1~400
	A_Location				: E_Location
	B_Location				: E_Location
	A_Done					: BOOL;
	B_Done					: BOOL;
END_STRUCT
END_TYPE

// ---- Library/10_Machine/18_HMI_Handshake/OLD_DUTs/DataCore/ST_SixRobotActionInfo.TcDUT
TYPE ST_SixRobotActionInfo :
STRUCT
	A_Done		:BOOL;
	B_Done		:BOOL;
END_STRUCT
END_TYPE

// ---- Library/10_Machine/18_HMI_Handshake/OLD_DUTs/DataCore/st_SixRobotAreaMove.TcDUT
TYPE st_SixRobotAreaMove :
STRUCT
	GET :BOOL;
	A_Area:	E_Location//A爪去放的位置
	B_Area:	E_Location//B爪去放的位置
	A_StorageInfor:INT
	B_StorageInfor:INT
	
	HandShake :st_HandshakeBase;
END_STRUCT
END_TYPE

// ---- Library/10_Machine/18_HMI_Handshake/OLD_DUTs/DataCore/st_SixRobotPTP.TcDUT
TYPE st_SixRobotPTP :
STRUCT
	A_AreaGet:	E_Location//A爪去取的位置
	B_AreaGet:	E_Location//B爪去取的位置
	A_StorageInfor:INT
	B_StorageInfor:INT
	
	A_AreaPut:	E_Location//A爪去放的位置
	B_AreaPut:	E_Location//B爪去放的位置
	A_StorageInfor:INT
	B_StorageInfor:INT
	
	HandShake :st_HandshakeBase;

END_STRUCT
END_TYPE

// ---- Library/10_Machine/18_HMI_Handshake/OLD_DUTs/DataCore/ST_WarehouseBack.TcDUT
TYPE ST_WarehouseBack :
STRUCT
		Info 	: ST_WarehouseBackInfo;
		Feeback : ST_WarehouseBackFeeback;
		Handshake	: ST_HandshakeBase;
END_STRUCT
END_TYPE

// ---- Library/10_Machine/18_HMI_Handshake/OLD_DUTs/DataCore/ST_WarehouseBackFeeback.TcDUT
TYPE ST_WarehouseBackFeeback :
STRUCT
	//提供圓帶上的針數
	AllocationInfo : ARRAY[0..40] OF st_AllocationData;
END_STRUCT
END_TYPE

// ---- Library/10_Machine/18_HMI_Handshake/OLD_DUTs/DataCore/ST_WarehouseBackInfo.TcDUT
TYPE ST_WarehouseBackInfo :
STRUCT
	//回傳那個圓帶回到哪個倉儲位置
	AllocationInfo : :ARRAY[0..40] OF st_AllocationData;
END_STRUCT
END_TYPE

// ---- Library/10_Machine/18_HMI_Handshake/OLD_DUTs/DataCore/ST_WarehouseGetBox.TcDUT
TYPE ST_WarehouseGetBox :
STRUCT
	//倉儲儲位
	StorageInfor	:INT;
	//盒子順序
	BoxOrder 		:INT;
END_STRUCT
END_TYPE

// ---- Library/10_Machine/18_HMI_Handshake/OLD_DUTs/DataCore/ST_ClampingToPlate.TcDUT
TYPE st_ClampingToPlate:
STRUCT
	//盒數
	NrOfBoxes				: INT;	// 1,2
	//放到哪裡
	TargetOfClipA			: INT;	// 0 : R1, 1: R2 or To plate index
	TargetOfClipB			: INT;	// 0 : R1, 1: R2 or To plate index
	//使用夾爪
	UseClibA				: BOOL;	//Clip A only work if True
	UseClibB				: BOOL;	//Clip B only work if True
	//從哪裡拿
	ClipAFrom				: INT; //0: 配好輸送帶。1: 同尺吋輸送帶
	ClipBFrom				: INT; //0: 配好輸送帶。1: 同尺吋輸帶
END_STRUCT
END_TYPE

// ---- Library/10_Machine/18_HMI_Handshake/OLD_DUTs/DataCore/st_DASCalibrationData.TcDUT
TYPE st_DASCalibrationData :
    STRUCT
        //出料手臂在配針區所有的校正位置
        OutRobotCore :ARRAY[0..99] OF st_OutRobotParameterCore;

        //配針手臂在圓帶的校正位置(第一盒的第一個 第二盒的第一個)
        AllocateCore :ARRAY[0..7] OF st_AllocateParameterCore;

        //配針手臂在圓盤的校正位置(第一盒的第一個 第二盒的第一個)
        TurnTableCore :ARRAY[0..7] OF st_AllocateParameterCore;

        // 成品區空盤電梯parameter //[0]=add position, [1]=empty position, [2]=plate gap
        OutAreaPlateElvatorPosition :ARRAY[0..2] OF st_OneDirectionCore;
        //成品區推出所有校正座標
        OutAreaPushMotoPosition :ARRAY[0..9] OF st_OneDirectionCore;
        //成品區電梯層架所有座標
        OutAreaElvatorPosition :ARRAY[0..5] OF st_OneDirectionCore;
        //分選區所有座標
        WarehouseMovePosition :ARRAY[0..3] OF st_OneDirectionCore;
        //所有馬達的內部參數
        ListMotoCore :ARRAY[0..10] OF st_ADSMotoCore;
        //所有馬達的內部移動參數
        ListMoveMoveCore :ARRAY[1..6] OF st_ADSMotoMoveCore;
        //出料區放盒的第一格位置 A 6-position B 6-position edit by johnson
        OutRobotfirstPosition :ARRAY[0..11] OF st_OutRobotParameterCore;
		//料架馬達的所有座標
		RackMotorPosition :ARRAY[0..9] OF st_OneDirectionCore;
    END_STRUCT
END_TYPE

// ---- Library/10_Machine/18_HMI_Handshake/OLD_DUTs/DataCore/ST_GetBoxData.TcDUT
TYPE ST_GetBoxData :
STRUCT
	//領盒資料
NeedleInfo					: ARRAY[0..200] OF ST_GetBoxInfo; 
//資料交握確認
	HandShake				: st_HandshakeBase;
END_STRUCT
 END_TYPE

// ---- Library/10_Machine/18_HMI_Handshake/OLD_DUTs/DataCore/ST_GetBoxInfo.TcDUT
TYPE ST_GetBoxInfo :
STRUCT
		//儲位
 		Storgerinfo		:INT; //1~400
		//軌道順序	
		Boxorder		:INT;//1~10
		//放的位置  
		Area  			:E_Location; 
END_STRUCT
 END_TYPE

// ---- Library/10_Machine/18_HMI_Handshake/OLD_DUTs/DataCore/ST_InformationExchange.TcDUT
TYPE ST_InformationExchange:
STRUCT
END_STRUCT
//配針領滿盒
NeedleFullBox						: ARRAY[0..300] OF ST_BoxGet
//配針換盒
NeedleChageBox						: 	ST_NeedleChageBox
//配針換圓帶
NeedleChageRotate					:	ST_NeedleChageRotate
//配針回倉
NeedleWarehouse						:	ARRAY[0..40] OF 		ST_NeedleWarehouse
//拔針領待拔針
NeedleRemoveBox						: ARRAY[0..30] OF ST_BoxGet
//拔針換盒
NeedleRemoveChageBox				:	ST_ NeedleChageBox
//拔針換圓帶
NeedleRemoveChageRotate				:	ST_NeedleChageRotate
//拔針回倉
NeedleRemoveWarehouse				:	ARRAY[0..40] OF 		ST_NeedleWarehouse
END_STRUCT
 END_TYPE

// ---- Library/10_Machine/18_HMI_Handshake/OLD_DUTs/DataCore/ST_MachineAdjust.TcDUT
TYPE ST_MachineAdjust :
STRUCT
	//回HOME 
	MachineHome          		: st_RegionHome;
	//手臂各區域點對點運動
	SixRobotPTP					: st_SixRobotPTP;
	//手臂各區域單動
	SixRobotAreaMove			: st_SixRobotAreaMove;
	//配針單動
	NeedleAction				: st_NeedleAction;
	//配針批量動作
	NeedleActionBatch			: st_NeedleActionBatch;
	//拔針批量動作
	NeedleRemoveActionBatch		: st_NeedleActionBatch;
	//料架站位移動
	BoxHookStationMove			: st_BoxHookStationMove;
	//層架站位移動
	LayerStationMove			: st_LayerStationMove;
	//勾盤站位移動
	PlateHookStationMove		: st_PlateHookStationMove;
	//出料手臂單動
	OutRobotMove				: st_OutRobotMove;
	//出料手臂連動
	OutRobotPTP					: st_OutRobotPTP;
	//圓帶站位移動
	AllocateStationMove			:st_AllocateStationMove;
	//圓盤站位移動
	TurnTableStationMove		:st_TurnTableStationMove;
END_STRUCT
END_TYPE

// ---- Library/10_Machine/18_HMI_Handshake/OLD_DUTs/DataCore/ST_MachineTask.TcDUT
TYPE ST_MachineTask :
STRUCT
	Feeding						: ST_Feeding;						//入料包含拍照
	Output						: ST_Output;						//出料
	Needle						: ST_Needle;						//配針資料提供
	NeedleRemove				: ST_NeedleRemove;					//拔針資料提供
	NeedleGetBox				: ST_GetBox;						//配針領料(滿盒)
	NeedleRemoveGetBox			: ST_GetBox;						//拔針領料(待拔針)
	NeedleChangeAllocate		: ST_ChangeAllocate;				//配針換圓帶
	NeedleRemoveChangeAllocate	: ST_ChangeAllocate;				//拔針換圓帶 
	WarehouseBack 				: ST_WarehouseBack;					//配針回倉
	WarehouseBackRemove 		: ST_WarehouseBack;					//拔針回倉
	SheepingPicture				: ST_SheepingPicture;				//出貨拍照
	AllocatePicture				: ST_SheepingPicture;				//圓帶拍照
	NeedleChangeBox				: ST9_ChangeBox; 					//配針換盒
	NeedleRemoveChangeBox		: ST9_ChangeBox;					//拔針換盒
	SixRobotWarehouseAction 	: ST_SixRobotAction,				//手臂倉儲動作				//手臂緩衝區動作
	Alarm						: ARRAY[0..999] OF ST_Alarm_Tmax;	//錯誤資訊
END_STRUCT
END_TYPE

// ---- Library/10_Machine/18_HMI_Handshake/OLD_DUTs/DataCore/ST_Needle.TcDUT
TYPE ST_Needle :
STRUCT
	//配針動作資料
		NeedleInfo							: ARRAY[0..2000] OF ST_AllocationJobBatchModeInfo; 
	//初始圓帶資料
		AllocationInfoData			 		:ARRAY[0..40] OF st_AllocationData;
	//空盒資料
		EmptyBoxCount						:INT;
	//滿盒資料
		FullboxCount						:INT;
	//鐵盤數資料
		PlateCount							:INT;
	//拍照位	1~6的鐵盤位加上鐵盤碼的位置
	PicturesLocation						: ARRAY[0..6] OF ST_PlateOrder;
	//出貨動作資料
		OutBoxMoveData 						: ST_ClampingToPlate;
	//資料交握確認
		HandShake							: ST_HandshakeBase;
END_STRUCT
END_TYPE

// ---- Library/10_Machine/18_HMI_Handshake/OLD_DUTs/DataCore/ST_NeedleChageBox.TcDUT
TYPE ST_NeedleChageBox :
STRUCT
	//確認是否要更換盒子
	CheckChageBox 	:BOOL; 
	//資料
	ST_NeedleChageBoxData : ARRAY[0..40] OF st_NeedleChageBoxData;
	//資料交握確認
	HandShake								: st_HandshakeBase;
END_STRUCT
END_TYPE

// ---- Library/10_Machine/18_HMI_Handshake/OLD_DUTs/DataCore/st_NeedleChageBoxData.TcDUT
TYPE st_NeedleChageBoxData :
STRUCT
	//圓帶位置
	AllocationNo 	:INT;
	//倉儲儲位
	StorageInfor	:INT;
	//盒子順序
	BoxOrder 		:INT;
END_STRUCT
END_TYPE

// ---- Library/10_Machine/18_HMI_Handshake/OLD_DUTs/DataCore/ST_NeedleWarehouse.TcDUT
TYPE ST_NeedleWarehouse :
STRUCT
	//提供回倉資料
	 NeedleWarehouseInfo 					:ST_NeedleWarehouseData;
	//資料交握確認
	HandShake								: st_HandshakeBase;
END_STRUCT
END_TYPE

// ---- Library/10_Machine/18_HMI_Handshake/OLD_DUTs/DataCore/ST_NeedleWarehouseData.TcDUT
TYPE ST_NeedleWarehouseData :
STRUCT
	ST_WarehouseData 	:ARRAY[0..40] OF st_WarehouseData;
END_STRUCT
END_TYPE

// ---- Library/10_Machine/18_HMI_Handshake/OLD_DUTs/DataCore/ST_SixRobotGetOrPut.TcDUT
TYPE ST_SixRobotGetOrPut :
STRUCT
	A_Clip_StorageInfor					:INT;
	A_Clip_BoxOrder						:INT;
	B_Clip_StorageInfor					:INT;
	B_Clip_BoxOrder						:INT;
	A_ActiveDone						:BOOL;
	B_ActiveDone						:BOOL;
	A_DataDone							:BOOL;
	B_DataDone							:BOOL;
END_STRUCT
END_TYPE

// ---- Library/10_Machine/18_HMI_Handshake/OLD_DUTs/DataCore/st_WarehouseData.TcDUT
TYPE st_WarehouseData :
STRUCT
	//圓帶位置
	AllocationNo 	:E_StationOrder;
	//放到哪裡
	AREA			:E_Location;
	//倉儲儲位
	StorageInfor	:INT;
	
END_STRUCT
END_TYPE

// ---- Library/10_Machine/18_HMI_Handshake/Service/DUTs/AllocateBatchMode/st_AllocateMoveAutoBatchMode_Ctrl.TcDUT
 TYPE st_AllocateMoveAutoBatchMode_Ctrl :
STRUCT
	bExecute			: BOOL; // Start Automode Turn Table process
	bReset				: BOOL; // Reset Automode Turn Table process
	bAbort				: BOOL; // Abort Automode Turn Table Process
	bOccupied			: BOOL;	
	bPause				: BOOL;
	bSimpleAllocation	: BOOL;
	AutoMode_AllocateMoveBatch 			:	 ST_AllocationJobBatchMode ;
END_STRUCT
END_TYPE

// ---- Library/10_Machine/18_HMI_Handshake/Service/DUTs/AllocateBatchMode/st_AllocateMoveAutoBatchMode_Status.TcDUT
TYPE st_AllocateMoveAutoBatchMode_Status :
STRUCT
	bBusy	: BOOL;
	bDone	: BOOL;
	bError	: BOOL;	
	bAborted : BOOL;
	ErrorID :UDINT;
	iIndex	: ARRAY[0..49] OF INT;
	Status   :STRING;
	uniqurErrorCode : STRING;
END_STRUCT
END_TYPE

// ---- Library/10_Machine/18_HMI_Handshake/Service/DUTs/AllocateBatchMode/st_Coordinate.TcDUT
TYPE st_Coordinate :
STRUCT
	X  : LREAL;
	Y  : LREAL;
	Rotate: LREAL;
END_STRUCT
END_TYPE

// ---- Library/10_Machine/18_HMI_Handshake/Service/DUTs/AllocateBatchMode/ST_Cylinders.TcDUT
TYPE
    ST_Cylinders :
    STRUCT
        Cylinder0 : REFERENCE TO FB_Cylinder;
        Cylinder1 : REFERENCE TO FB_Cylinder;
        Cylinder2 : REFERENCE TO FB_Cylinder;
        Cylinder3 : REFERENCE TO FB_Cylinder;
    END_STRUCT
END_TYPE

// ---- Library/10_Machine/18_HMI_Handshake/Service/DUTs/AllocateBatchMode/st_RoundBeltAutoSingleMove_Ctrl.TcDUT
TYPE st_RoundBeltAutoSingleMove_Ctrl :
STRUCT	
		bExecute                  :BOOL;                     
        bReset                    :BOOL;                     
        bAbort                    :BOOL;           
        uiStation				  :UINT;  
		uiLatch					  :UINT;     
        Timeout					  :TIME := T#3S; 
		bOccupied				  :BOOL;
		bSendPressBox			  :BOOL;	
END_STRUCT
END_TYPE

// ---- Library/10_Machine/18_HMI_Handshake/Service/DUTs/AllocateBatchMode/U_Cylinders.TcDUT
TYPE
    U_Cylinders :
    UNION
        Cylinders   : REFERENCE TO ARRAY[0..3] OF FB_Cylinder;
        stCylinders : ST_Cylinders;
    END_UNION
END_TYPE

// ---- Library/10_Machine/18_HMI_Handshake/Service/DUTs/ST_HMI_Handshake.TcDUT
TYPE
    ST_HMI_Handshake :
    STRUCT
       //========單動一行程============
	// one process use
    //配針單動資料結構
    AllocateMoveStructure : REFERENCE TO st_ads_AllocateMoveStructure;
	//拔針單動資料結構
    AllocateMoveStructure_Reverse : REFERENCE TO st_ads_AllocateMoveStructure;     
    //空盒手臂單動資料結構
    EmptyRobotToTurnTableMove : REFERENCE TO st_ads_OneAxisMoveWithPosition;
    //圓帶單動一行程
    AllocateCircleMove : REFERENCE TO st_AllocateCircleMoveStructure;
    //圓盤單動一行程
    TurnTableMove : REFERENCE TO st_ads_OneAxisMoveWithPosition;
//    //軸還原預設狀態
//    AxesControl : REFERENCE TO ARRAY[0..10] OF st_AxisControl;
    //機台還原預設狀態
    MachineReset : REFERENCE TO st_ads_MachineReset;
    //Empty
    RareFullBoxPush : REFERENCE TO st_ads_OutRobtToPlateMove;
		// Move Allocate robot to needling position
	AllocationRobotNeedlingMove : REFERENCE TO st_AllocateRobotNeedlingMove;

//==============自動模式=========================

    //AutoModeUse*-------自動模式圓帶單動
    AutoMode_AllocateCircleMove : REFERENCE TO st_AllocateCircleMoveStructure;
    //AutoModeUse*-------手臂倉儲位置移動
    AutoMode_RobotWarehouseMove : REFERENCE TO st_AutoSixAxisWarehouseParameter;
    //AutoModeUse*-------手臂絕對位置移動
    AutoMode_RobotAbsMove : REFERENCE TO st_AutoSixAxisAbsMoveParameter;
    //AutoModeUse*-------空盒取料移動
    AutoMode_EmptyBoxMove : REFERENCE TO st_AutoMode_ClampingBoxesJob;
    //AutoModeUse*-------圓盤移動
    AutoMode_TurnTableMOve : REFERENCE TO st_ads_OneAxisMoveWithPosition;
    //AutoModeUse--------配針
    AutoMode_AllocateMove : REFERENCE TO st_AutoMode_AllocatingJob;
	 //AutoModeUse--------拔針
    AutoMode_AllocateMove_Reverse : REFERENCE TO st_AutoMode_AllocatingJob;
	//AutoModeUse--------配針batch mode
	AutoMode_AllocateBatchMode	: REFERENCE TO ST_AllocationJobBatchMode;
	//AutoModeUse--------拔針batch mode
	AutoMode_AllocateBatchMode_Reverse	: REFERENCE TO ST_AllocationJobBatchMode;
	//AutoModeSimpleAllocation_Batch
	AutoMode_SimpleAllocation_Batch		: REFERENCE TO ST_AllocationJobBatchMode;
    //AutoMdeUse---------散針放盒
    AutoMode_RareBoxMove : REFERENCE TO st_AutoMode_ClampingBoxesJob;
    //AutoMdeUse---------出貨放盒單動
    AutoMode_OutBoxMove : REFERENCE TO st_AutoMode_ClampingToPlate;
	//AutoMdeUse---------拔針放盒自動模式
    AutoMode_BoxMoveReverse : REFERENCE TO st_AutoMode_ClampingBoxesJob;
    //倉儲分選區移動,移動位置列表需延伸此陣列取得 WarehouseMovePosition :ARRAY[0..3] OF st_OneDirectionCore;
    AutoMode_WarehouseMove : REFERENCE TO st_ads_OneAxisMoveWithPosition;
    //AutoModeUse------手臂區域移動_FeedIn conveyor
	AutoMode_RobotRegionMove_FeedInConveyor		: REFERENCE TO ST_AutoMode_RobotRegionMove;
	//AutoModeUse------手臂區域移動_AllocatedConveyor
	AutoMode_RobotRegionMove_AllocatedConveyor		: REFERENCE TO ST_AutoMode_RobotRegionMove;
	//AutoModeUse------手臂區域移動_Pullout conveyor
	AutoMode_RobotRegionMove_PullOutConveyor		: REFERENCE TO ST_AutoMode_RobotRegionMove;
	//AutoModeUse------手臂區域移動_Buffer area
	AutoMode_RobotRegionMove_BufferArea		: REFERENCE TO ST_AutoMode_RobotRegionMove;
	//AutoModeUse------手臂區域移動_RoundBelt
	AutoMode_RobotRegionMove_RoundBelt		: REFERENCE TO ST_AutoMode_RobotRegionMove;
   //AutoMode MoveConveyorJob------定時移動輸送帶
    AutoMode_MoveConveyorJob : REFERENCE TO st_MoveConveyorJob;
	// Automode Feedin empty box with robot 
	AutoMode_FeedInEmptyBoxWithRobot : REFERENCE TO ST_AutoMode_FeedInEmptyBox; // Automode : Feedin empty box with robot from Warehouse and Pullout convenyor
	// Automode Reload RoundBelt box with robot
	AutoMode_ReloadRoundBeltBoxWithRobot : REFERENCE TO ST_AutoMode_ReloadRoundBeltBox; // Automode : Reload RoundBelt box with robot from warehouse
	//AutoMode UpperFeedInConveyor
	AutoMode_UpperFeedInConveyor : REFERENCE TO ST_Auto_UpperFeedInConveyor;
	//AutoModeUse------倉儲馬達搭配手臂移動
    AutoMode_WarehouseMotoWithRobotMove : REFERENCE TO st_AutoSixAxisWarehouseParameter;
    //SimpleAllocate Autode-----簡易配針
	AutoMode_SimpleAllocate    : REFERENCE TO ST_AutoMode_SimpleAllocateHandShake; // AutoMode Simple Allocate
    AutoMode_PullOutConveyor   : REFERENCE TO ST_AutoPullOutConveyor; // AutoMode PullOut Conveyor
    //AutoModeUse----------錯誤通知  Host To PLC
    AutoMode_ErrorHandle : REFERENCE TO st_Alarm;
    //Alarm report	----------錯誤通知 PLC to Host
    AlarmAllocation : REFERENCE TO ARRAY[0..999] OF ST_Alarm_Tmax;
	//AutoMode Use------ShippingGoodV2		20250304 Min
	AutoMode_AddBoxes	: REFERENCE TO ST_AutoAddsBoxes;
    //=================TwinCat Memory============
    //TwinCatMemory				:st_TwinCatMemory;
    //=================全局Home===================

    MachineHome          : REFERENCE TO st_RegionHome; // Machine all units home command
    StorageRegionHome    : REFERENCE TO st_RegionHome;
    AllocationRegionHome : REFERENCE TO st_RegionHome;
    FGARegionHome        : REFERENCE TO st_RegionHome;

    //===============手自動=======================
    StorageRegionMode : REFERENCE TO ST_Mode;
    AllocationRegion  : REFERENCE TO ST_Mode;
    FGARegionMode     : REFERENCE TO ST_Mode;
    MachineMode       : REFERENCE TO ST_Mode;
	
    // Operation Pannel Status
    OpPannel_Status : REFERENCE TO ST_OpPannelStatus; //PLC -> HMI
    OpPannel_Ctrl   : REFERENCE TO ST_OpPannelStatus; // HMI -> PLC

	//20250425 addon
	//Machine state
//	MachineState : REFERENCE TO E_MachineState;
	
	FanucRobot_General               : REFERENCE TO ST_FanucRobotGeneralCtrl;
	
	//AutoModeUse------倉儲小手臂ABS 移動
	AutoMode_ShippingRobot_Left            : REFERENCE TO ST_AutoMode_ShippingRobot_MoveAbs;
	//AutoModeUse------倉儲小手臂ABS 移動
	AutoMode_ShippingRobot_Right           :REFERENCE TO  ST_AutoMode_ShippingRobot_MoveAbs;
	//AutoModeUse------倉儲小手臂ABS 移動
	AutoMode_ShippingRobot_TransmitCVEnd    : REFERENCE TO ST_AutoMode_ShippingRobot_MoveAbs;
	//AutoModeUse------同尺寸拍照			
	AutoMode_SameSizeCVCamera				: REFERENCE TO ST_AutoMode_TransCVCamera;
	//AutoModeUse------不同尺寸拍照	
	AutoMode_DifferentCVCamera				: REFERENCE TO ST_AutoMode_TransCVCamera;


    END_STRUCT
END_TYPE

// ---- Library/10_Machine/19_Device/EL1889/ST_EbusDI16.TcDUT
TYPE ST_EbusDI16 :
    STRUCT
        DI1  AT %I* :BIT;
        DI2  AT %I* :BIT;
        DI3  AT %I* :BIT;
        DI4  AT %I* :BIT;
        DI5  AT %I* :BIT;
        DI6  AT %I* :BIT;
        DI7  AT %I* :BIT;
        DI8  AT %I* :BIT;
        DI9  AT %I* :BIT;
        DI10 AT %I* :BIT;
        DI11 AT %I* :BIT;
        DI12 AT %I* :BIT;
        DI13 AT %I* :BIT;
        DI14 AT %I* :BIT;
        DI15 AT %I* :BIT;
        DI16 AT %I* :BIT;
    END_STRUCT
END_TYPE

// ---- Library/10_Machine/19_Device/EL1889/ST_EbusInputModule.TcDUT
TYPE
    ST_EbusInputModule :
    STRUCT
        EL1889_01 : ST_EbusDI16;
        EL1889_02 : ST_EbusDI16;
        EL1889_03 : ST_EbusDI16;
        EL1889_04 : ST_EbusDI16;
        EL1889_05 : ST_EbusDI16;
        EL1889_06 : ST_EbusDI16;
        EL1889_07 : ST_EbusDI16;
        EL1889_08 : ST_EbusDI16;
        EL1889_09 : ST_EbusDI16;
        EL1889_10 : ST_EbusDI16;
        EL1889_11 : ST_EbusDI16;
    END_STRUCT
END_TYPE

// ---- Library/10_Machine/19_Device/EL1889/ST_InputTable.TcDUT
TYPE
    ST_InputTable :
    STRUCT
        bUpCV_BoxArrived_Sensor                       : BIT; //X6.0
        bUpCV_Block1Detect_Sensor                     : BIT; //X6.1
        bUpCV_Block2Detect_Sensor                     : BIT; //X6.2
        bUpCV_Block3Detect_Sensor                     : BIT; //X6.3
        bUpCV_ReLoadDetect_Sensor                     : BIT; //X6.4
        bUpCV_Block1_RearSensor                       : BIT; //X6.5
        bUpCV_Block2_RearSensor                       : BIT; //X6.6
        bUpCV_Block3_RearSensor                       : BIT; //X6.7
        bLowCV_BoxArrived_Sensor                      : BIT; //X6.8
        bLowCV_Block1Detect_Sensor                    : BIT; //X6.9
        bLowCV_Block2Detect_Sensor                    : BIT; //X6.10
        bLowCV_Block1_RearSensor                      : BIT; //X6.11
        bLowCV_Block2_RearSensor                      : BIT; //X6.12
        bLowCV_2ndBoxGap_Sensor                       : BIT; //X6.13
        spare15                                       : BIT; //X6.14
        spare16                                       : BIT; //X6.15
        bUpCV_DiameterHoriz_FrontSensor               : BIT; //X7.0
        bUpCV_DiameterHoriz_RearSensor                : BIT; //X7.1
        bUpCV_DiameterVert_FrontSensor                : BIT; //X7.2
        bUpCV_DiameterVert_RearSensor                 : BIT; //X7.3
        spare21                                       : BIT; //X7.4
        spare22                                       : BIT; //X7.5
        spare23                                       : BIT; //X7.6
        spare24                                       : BIT; //X7.7
        spare25                                       : BIT; //X7.8
        spare26                                       : BIT; //X7.9
        bStorage_AirPressure_Ready                    : BIT; //X7.10
        bStorage_EstopPb                              : BIT; //X7.11
        bStorage_StartPb                              : BIT; //X7.12
        bStorage_StopPb                               : BIT; //X7.13
        bStorage_ResetPb                              : BIT; //X7.14
        spare32				                          : BIT; //X7.15
        bStackPush_DCMotor_PosLimit                   : BIT; //X9.0
        bStackPush_DCMotor_NegLimit                   : BIT; //X9.1
        bStackPush_Pusher_FrontSensor                 : BIT; //X9.2
        bStackPush_Pusher_RearSensor                  : BIT; //X9.3
        bStorage_StackPushPb                          : BIT; //X9.4
        Spare38                                       : BIT; //X9.5
        Spare39                                       : BIT; //X9.6
        Spare40                                       : BIT; //X9.7
        bPullOutCV_AsideEntry_Sensor                  : BIT; //X9.8
        bPullOutCV_AsideExit_Sensor                   : BIT; //X9.9
        bPullOutCV_Aside2ndBoxGap_Sensor              : BIT; //X9.10
        bPullOutCV_BsideEntry_Sensor                  : BIT; //X9.11
        bPullOutCV_BsideExit_Sensor                   : BIT; //X9.12
        bPullOutCV_Bside2ndBoxGap_Sensor              : BIT; //X9.13
        bPullOutCV_AsideBlock_RearSensor              : BIT; //X9.14
        bPullOutCV_BsideBlock_RearSensor              : BIT; //X9.15
        bSafetyDoor1                                  : BIT; //X10.0
        bSafetyDoor2                                  : BIT; //X10.1
        bSafetyDoor14                                 : BIT; //X10.2
        Spare52                                       : BIT; //X10.3
        bSafetyDoor13                                 : BIT; //X10.4
        bSafetyDoor12                                 : BIT; //X10.5
        bSafetyDoor11                                 : BIT; //X10.6
        bSafetyDoor10                                 : BIT; //X10.7
        bSafetyDoor9                                  : BIT; //X10.8
        spare58                                       : BIT; //X10.9
        spare59                                       : BIT; //X10.10
        spare60                                       : BIT; //X10.11
        spare61                                       : BIT; //X10.12
        spare62                                       : BIT; //X10.13
        bPullOutCV_FwdPb                              : BIT; //X10.14
        bPullOutCV_RevPb                              : BIT; //X10.15
        bAllocateRobot_LeftVert1_HighSensor           : BIT; //X0.0
        bAllocateRobot_LeftVert1_LowSensor            : BIT; //X0.1
        bAllocateRobot_LeftVert2_HighSensor           : BIT; //X0.2
        bAllocateRobot_LeftVert2_LowSensor            : BIT; //X0.3
        bAllocateRobot_RightVert1_HighSensor          : BIT; //X0.4
        bAllocateRobot_RightVert1_LowSensor           : BIT; //X0.5
        bAllocateRobot_RightVert2_HighSensor          : BIT; //X0.6
        bAllocateRobot_RightVert2_LowSensor           : BIT; //X0.7
        bRoundBelt_ChangeZoneA2Detect_Sensor          : BIT; //X0.8
        bRoundBelt_ChangeZoneA3Detect_Sensor          : BIT; //X0.9
        bRoundBelt_ChangeZonePlug_FrontSensor         : BIT; //X0.10
        bRoundBelt_ChangeZonePlug_RearSensor          : BIT; //X0.11
        bRoundBelt_WorkZoneQ1Detect_Sensor            : BIT; //X0.12
        bRoundBelt_WorkZoneQ2Detect_Sensor            : BIT; //X0.13
        bRoundBelt_WorkZonePlug_FrontSensor           : BIT; //X0.14
        bRoundBelt_WorkZonePlug_RearSensor            : BIT; //X0.15
        bRoundBelt_WorkZonePress_RearSensor           : BIT; //X1.0
        bTempZoneA_Sensor                             : BIT; //X1.1
        bTempZoneB_Sensor                             : BIT; //X1.2
        bTempZoneC_Sensor                             : BIT; //X1.3
        bTempZoneD_Sensor                             : BIT; //X1.4
        bTurnTable_Press_RearSensor                   : BIT; //X1.5
        bTurnTable_R1Detect_Sensor                    : BIT; //X1.6
        bTurnTable_R2Detect_Sensor                    : BIT; //X1.7
        bTurnTable_I2Detect_Sensor                    : BIT; //X1.8
        bTurnTable_I1Detect_Sensor                    : BIT; //X1.9
        bOutRobot_Xaxis_PosLimit                      : BIT; //X1.10
        bOutRobot_Xaxis_HomeSensor                    : BIT; //X1.11
        bOutRobot_Xaxis_NegLimit                      : BIT; //X1.12
        bOutRobot_Yaxis_PosLimit                      : BIT; //X1.13
        bOutRobot_Yaxis_HomeSensor                    : BIT; //X1.14
        bOutRobot_Yaxis_NegLimit                      : BIT; //X1.15
        bOutRobot_AsideVert_HighSensor                : BIT; //X2.0
        bOutRobot_AsideVert_LowSensor                 : BIT; //X2.1
        bOutRobot_BsideVert_HighSensor                : BIT; //X2.2
        bOutRobot_BsideVert_LowSensor                 : BIT; //X2.3
        bOutRobot_AsideClamp_RearSensor               : BIT; //X2.4
        bOutRobot_BsideClamp_RearSensor               : BIT; //X2.5
        spare103                                      : BIT; //X2.6
        bSafetyDoor5			                      : BIT; //X2.7
        spare105                                      : BIT; //X2.8
        bSafetyDoor3                                  : BIT; //X2.9
        bAllocate_Electrical_Cabinet_SafetyDoor       : BIT; //X2.10
        bAllocate_AirPressure_Ready                   : BIT; //X2.11
        bAllocate_StartPb                             : BIT; //X2.12
        bAllocate_StopPb                              : BIT; //X2.13
        bAllocate_ResetPb                             : BIT; //X2.14
        bAllocate_EStopPb                             : BIT; //X2.15
        bSameSizeCV_BoxNearStorageSensor              : BIT; //X3.0
        bDifferentSizeCV_BoxDetect7_Sensor            : BIT; //X3.1
        bDifferentSizeCV_BoxDetect6_Sensor            : BIT; //X3.2
        bDifferentSizeCV_BoxDetect5_Sensor            : BIT; //X3.3
        bDifferentSizeCV_BoxDetect4_Sensor            : BIT; //X3.4
        bTransmit_CamaraHorizDifferentSizeSide_Sensor : BIT; //X3.5
        bTransmit_CamaraHorizSameSizeSide_Sensor      : BIT; //X3.6
        bDifferentSizeCV_BoxDetect3_Sensor            : BIT; //X3.7
        bDifferentSizeCV_BoxDetect2_Sensor            : BIT; //X3.8
        bDifferentSizeCV_BoxDetect1_Sensor            : BIT; //X3.9
        bDifferentSizeCV_BoxNearShippingSensor        : BIT; //X3.10
        bSameSizeCV_BoxDetect6_Sensor                 : BIT; //X3.11
        bSameSizeCV_BoxDetect5_Sensor                 : BIT; //X3.12
        bSameSizeCV_BoxDetect4_Sensor                 : BIT; //X3.13
        Spare127                                      : BIT; //X3.14
        bSameSizeCV_BoxDetect3_Sensor                 : BIT; //X3.15
        bRoundBelt_TransmitCVZonePlug_RearSensor      : BIT; //X8.0
        bRoundBelt_TransmitCVZonePlug_FrontSensor     : BIT; //X8.1
        bRoundBelt_Axis_HomeSensor                    : BIT; //X8.2
        spare132	                                  : BIT; //X8.3
        bSafetyDoor7   		                          : BIT; //X8.4
        bSafetyDoor8           		                  : BIT; //X8.5
        bShippingRobot_ElectricalCabinet_SafetyDoor    : BIT; //X8.6
        bSafetyDoor6                       		      : BIT; //X8.7
        spare137	                                  : BIT; //X8.8
        bTurnTable_Axis_HomeSensor                    : BIT; //X8.9
        bAllocateRobot_Xaxis_PosLimit                 : BIT; //X8.10
        bAllocateRobot_Xaxis_NegLimit                 : BIT; //X8.11
        bSafetyDoor4                                  : BIT; //X8.12
        bSameSizeCV_BoxDetect1_Sensor                 : BIT; //X8.13
        bSameSizeCV_BoxNearShippingSensor             : BIT; //X8.14
        bSameSizeCV_BoxDetect2_Sensor                 : BIT; //X8.15
        bDifferentCV_Block_RearSensor                 : BIT; //X11.0
        bSameSizeCVBlock1_RearSensor                  : BIT; //X11.1
        bSameSizeCVBlock2_RearSensor                  : BIT; //X11.2
        spare148                                      : BIT; //X11.3
        spare149                                      : BIT; //X11.4
        spare150                                      : BIT; //X11.5
        spare151                                      : BIT; //X11.6
        spare152                                      : BIT; //X11.7
        spare153                                      : BIT; //X11.8
        spare154                                      : BIT; //X11.9
        spare155                                      : BIT; //X11.10
        spare156                                      : BIT; //X11.11
        spare157                                      : BIT; //X11.12
        spare158                                      : BIT; //X11.13
        spare159                                      : BIT; //X11.14
        spare160                                      : BIT; //X11.15
        bShipping_NgCV1_Sensor                        : BIT; //X4.0
        bShipping_NgCV2_Sensor                        : BIT; //X4.1
        spare163                                      : BIT; //X4.2
        spare164                                      : BIT; //X4.3
        spare165                                      : BIT; //X4.4
        spare166                                      : BIT; //X4.5
        spare167                                      : BIT; //X4.6
        spare168                                      : BIT; //X4.7
        spare169                                      : BIT; //X4.8
        spare170                                      : BIT; //X4.9
        spare171                                      : BIT; //X4.10
        spare172                                      : BIT; //X4.11
        spare173                                      : BIT; //X4.12
        spare174                                      : BIT; //X4.13
        spare175                                      : BIT; //X4.14
        spare176                                      : BIT; //X4.15
    END_STRUCT
END_TYPE

// ---- Library/10_Machine/19_Device/EL1889/ST_InputTable_Mitsubishi.TcDUT
TYPE
    ST_InputTable_Mitsubishi :
    STRUCT
        X6  : uni_IntToBool;
        X7  : uni_IntToBool;
        X9  : uni_IntToBool;
        X10 : uni_IntToBool;
        X0  : uni_IntToBool;
        X1  : uni_IntToBool;
        X2  : uni_IntToBool;
        X3  : uni_IntToBool;
        X8  : uni_IntToBool;
        X11 : uni_IntToBool;
        X4  : uni_IntToBool;
    END_STRUCT
END_TYPE

// ---- Library/10_Machine/19_Device/EL1889/uni_InputModule.TcDUT
TYPE
    uni_InputModule :
    UNION
        stEbusDI : ST_EbusInputModule;       // Input table defined based on module allocation.
        stDI     : ST_InputTable;            // Input table defined based on variable names.
        stDIList : ST_InputTable_Mitsubishi; //Input table defined based on Mitsubishi PLC conventions.
    END_UNION
END_TYPE

// ---- Library/10_Machine/19_Device/EL2889/ST_EbusDO16.TcDUT
TYPE ST_EbusDO16 :
    STRUCT
        DO1  AT %Q* :BIT;
        DO2  AT %Q* :BIT;
        DO3  AT %Q* :BIT;
        DO4  AT %Q* :BIT;
        DO5  AT %Q* :BIT;
        DO6  AT %Q* :BIT;
        DO7  AT %Q* :BIT;
        DO8  AT %Q* :BIT;
        DO9  AT %Q* :BIT;
        DO10 AT %Q* :BIT;
        DO11 AT %Q* :BIT;
        DO12 AT %Q* :BIT;
        DO13 AT %Q* :BIT;
        DO14 AT %Q* :BIT;
        DO15 AT %Q* :BIT;
        DO16 AT %Q* :BIT;
    END_STRUCT
END_TYPE

// ---- Library/10_Machine/19_Device/EL2889/ST_EbusOutputModule.TcDUT
TYPE ST_EbusOutputModule :
    STRUCT
        EL2889_01 :ST_EbusDO16;
        EL2889_02 :ST_EbusDO16;
        EL2889_03 :ST_EbusDO16;
        EL2889_04 :ST_EbusDO16;
        EL2889_05 :ST_EbusDO16;
        EL2889_06 :ST_EbusDO16;
        EL2889_07 :ST_EbusDO16;
        EL2889_08 :ST_EbusDO16;
        EL2889_09 :ST_EbusDO16;
        EL2889_10 :ST_EbusDO16;
    END_STRUCT
END_TYPE

// ---- Library/10_Machine/19_Device/EL2889/ST_OutputTable.TcDUT
TYPE
    ST_OutputTable :
    STRUCT
        bUpCV_FeedInPress1_Valve                   : BIT; //Y4.0
        bUpCV_FeedInPress2_Valve                   : BIT; //Y4.1
        bUpCV_DiameterPress_Valve                  : BIT; //Y4.2
        bUpCV_CamaraPress1_Valve                   : BIT; //Y4.3
        bUpCV_CamaraPress2_Valve                   : BIT; //Y4.4
        bUpCV_CamaraPress3_Valve                   : BIT; //Y4.5
        bUpCV_CamaraPress4_Valve                   : BIT; //Y4.6
        bUpCV_Block1_Up_Valve                      : BIT; //Y4.7
        bUpCV_Block1_Down_Valve                    : BIT; //Y4.8
        bUpCV_Block2_Up_Valve                      : BIT; //Y4.9
        bUpCV_Block2_Down_Valve                    : BIT; //Y4.10
        bUpCV_Block3_Up_Valve                      : BIT; //Y4.11
        bUpCV_Block3_Down_Valve                    : BIT; //Y4.12
        Spare14                                    : BIT; //Y4.13
        Spare15                                    : BIT; //Y4.14
        Spare16                                    : BIT; //Y4.15
        bWareHouseCV10_Fwd                         : BIT; //Y5.0
        bWareHouseCV10_Rev                         : BIT; //Y5.1
        bWareHouseCV9_Fwd                          : BIT; //Y5.2
        bWareHouseCV9_Rev                          : BIT; //Y5.3
        bWareHouseCV8_Fwd                          : BIT; //Y5.4
        bWareHouseCV8_Rev                          : BIT; //Y5.5
        bWareHouseCV7_Fwd                          : BIT; //Y5.6
        bWareHouseCV7_Rev                          : BIT; //Y5.7
        bWareHouseCV6_Fwd                          : BIT; //Y5.8
        bWareHouseCV6_Rev                          : BIT; //Y5.9
        bWareHouseCV5_Fwd                          : BIT; //Y5.10
        bWareHouseCV5_Rev                          : BIT; //Y5.11
        bWareHouseCV4_Fwd                          : BIT; //Y5.12
        bWareHouseCV4_Rev                          : BIT; //Y5.13
        bWareHouseCV3_Fwd                          : BIT; //Y5.14
        bWareHouseCV3_Rev                          : BIT; //Y5.15
        bWareHouseCV2_Fwd                          : BIT; //Y6.0
        bWareHouseCV2_Rev                          : BIT; //Y6.1
        bWareHouseCV1_Fwd                          : BIT; //Y6.2
        bWareHouseCV1_Rev                          : BIT; //Y6.3
        bWareHouseCV20_Fwd                         : BIT; //Y6.4
        bWareHouseCV20_Rev                         : BIT; //Y6.5
        bWareHouseCV19_Fwd                         : BIT; //Y6.6
        bWareHouseCV19_Rev                         : BIT; //Y6.7
        bWareHouseCV18_Fwd                         : BIT; //Y6.8
        bWareHouseCV18_Rev                         : BIT; //Y6.9
        bWareHouseCV17_Fwd                         : BIT; //Y6.10
        bWareHouseCV17_Rev                         : BIT; //Y6.11
        bWareHouseCV16_Fwd                         : BIT; //Y6.12
        bWareHouseCV16_Rev                         : BIT; //Y6.13
        bWareHouseCV15_Fwd                         : BIT; //Y6.14
        bWareHouseCV15_Rev                         : BIT; //Y6.15
        bWareHouseCV14_Fwd                         : BIT; //Y7.0
        bWareHouseCV14_Rev                         : BIT; //Y7.1
        bWareHouseCV13_Fwd                         : BIT; //Y7.2
        bWareHouseCV13_Rev                         : BIT; //Y7.3
        bWareHouseCV12_Fwd                         : BIT; //Y7.4
        bWareHouseCV12_Rev                         : BIT; //Y7.5
        bWareHouseCV11_Fwd                         : BIT; //Y7.6
        bWareHouseCV11_Rev                         : BIT; //Y7.7
        bUpCV_Fwd                                  : BIT; //Y7.8
        bUpCV_Rev                                  : BIT; //Y7.9
        bLowCV_Fwd                                 : BIT; //Y7.10
        bLowCV_Rev                                 : BIT; //Y7.11
        bPullOutCV_A_Fwd                           : BIT; //Y7.12
        bPullOutCV_A_Rev                           : BIT; //Y7.13
        bPullOutCV_B_Fwd                           : BIT; //Y7.14
        bPullOutCV_B_Rev                           : BIT; //Y7.15
        bUpCV_DiameterHoriz_Extend_Valve           : BIT; //Y8.0
        bUpCV_DiameterHoriz_Retract_Valve          : BIT; //Y8.1
        bUpCV_DiameterVert_Valve                   : BIT; //Y8.2
        bUpCV_DiameterClamp_Close_Valve            : BIT; //Y8.3
        bUpCV_DiameterClamp_Open_Valve             : BIT; //Y8.4
        bStackPush_Valve                           : BIT; //Y8.5
        bCamara_Blow                               : BIT; //Y8.6
        Spare72                                    : BIT; //Y8.7
        bStorage_StartPbLamp                       : BIT; //Y8.8
        bStorage_StopPbLamp                        : BIT; //Y8.9
        bStorage_ResetPbLamp                       : BIT; //Y8.10
        bStorage_StackPushPbLamp                   : BIT; //Y8.11
        bStorage_EleBoxLight                       : BIT; //Y8.12
        bPullOutCV_FwdPbLamp                       : BIT; //Y8.13
        bPullOutCV_RevPbLamp                       : BIT; //Y8.14
        bStorage_FanucRobotPower                   : BIT; //Y8.15
        bStorage_SingleTower_BlueLamp              : BIT; //Y10.0
        bStorage_SingleTower_RedLamp           	   : BIT; //Y10.1
        bStorage_SingleTower_YellowLamp            : BIT; //Y10.2
        bStorage_SingleTower_GreenLamp             : BIT; //Y10.3
        bStorage_Buzzer                            : BIT; //Y10.4
        Spare86                                    : BIT; //Y10.5
        Spare87                                    : BIT; //Y10.6
        bStorage_AreaLight                         : BIT; //Y10.7
        bPullOutCV_AsidePress1_Valve               : BIT; //Y10.8
        bPullOutCV_AsidePress2_Valve               : BIT; //Y10.9
        bPullOutCV_AsideBlock_Valve                : BIT; //Y10.10
        bPullOutCV_BsidePress1_Valve               : BIT; //Y10.11
        bPullOutCV_BsidePress2_Valve               : BIT; //Y10.12
        bPullOutCV_BsideBlock_Valve                : BIT; //Y10.13
        Spare95                                    : BIT; //Y10.14
        Spare96                                    : BIT; //Y10.15
        bLowCV_Press1_Valve                        : BIT; //Y11.0
        bLowCV_Press2_Valve                        : BIT; //Y11.1
        bLowCV_Press3_Valve                        : BIT; //Y11.2
        bLowCV_Press4_Valve                        : BIT; //Y11.3
        bLowCV_Block1_Up_Valve                     : BIT; //Y11.4
        bLowCV_Block1_Down_Valve                   : BIT; //Y11.5
        bLowCV_Block2_Up_Valve                     : BIT; //Y11.6
        bLowCV_Block2_Down_Valve                   : BIT; //Y11.7
        Spare105                                   : BIT; //Y11.8
        Spare106                                   : BIT; //Y11.9
        Spare107                                   : BIT; //Y11.10
        Spare108                                   : BIT; //Y11.11
        Spare109                                   : BIT; //Y11.12
        Spare110                                   : BIT; //Y11.13
        Spare111                                   : BIT; //Y11.14
        Spare112                                   : BIT; //Y11.15
        bAllocateRobot_LeftVert1_Valve             : BIT; //Y0.0
        bAllocateRobot_LeftVert2_Valve             : BIT; //Y0.1
        bAllocateRobot_RightVert1_Valve            : BIT; //Y0.2
        bAllocateRobot_RightVert2_Valve            : BIT; //Y0.3
        bAllocateRobot_LeftClamp1_Close_Valve      : BIT; //Y0.4
        bAllocateRobot_LeftClamp1_Open_Valve       : BIT; //Y0.5
        bAllocateRobot_LeftClamp2_Close_Valve      : BIT; //Y0.6
        bAllocateRobot_LeftClamp2_Open_Valve       : BIT; //Y0.7
        bAllocateRobot_RightClamp1_Close_Valve     : BIT; //Y0.8
        bAllocateRobot_RightClamp1_Open_Valve      : BIT; //Y0.9
        bAllocateRobot_RightClamp2_Close_Valve     : BIT; //Y0.10
        bAllocateRobot_RightClamp2_Open_Valve      : BIT; //Y0.11
        bRoundBelt_WorkZone_Press_Valve            : BIT; //Y0.12
        bRoundBelt_WorkZone_Plug_Valve             : BIT; //Y0.13
        bRoundBelt_ChargeZone_Plug_Valve           : BIT; //Y0.14
        bRoundBelt_TransmitCVZone_Plug_Valve       : BIT; //Y0.15
        bOutRobot_AsideVert_Valve                  : BIT; //Y1.0
        bOutRobot_BsideVert_Valve                  : BIT; //Y1.1
        bOutRobot_AsideClamp_Close_Valve           : BIT; //Y1.2
        bOutRobot_AsideClamp_Open_Valve            : BIT; //Y1.3
        bOutRobot_BsideClamp_Close_Valve           : BIT; //Y1.4
        bOutRobot_BsideClamp_Open_Valve            : BIT; //Y1.5
        bTransmitCV_CamaraHorizDifferentSide_Valve  : BIT; //Y1.6
        bTransmitCV_CamaraHorizSameSizeSide_Valve: BIT; //Y1.7
        bDifferentSizeCV_Press2_Valve              : BIT; //Y1.8
        bDifferentSizeCV_Press1_Valve              : BIT; //Y1.9
        bDifferentSizeCV_Block1_Valve              : BIT; //Y1.10
        bSameSizeCV_Press4_Valve                   : BIT; //Y1.11
        bSameSizeCV_Press3_Valve                   : BIT; //Y1.12
        bSameSizeCV_Press2_Valve                   : BIT; //Y1.13
        bSameSizeCV_Press1_Valve                   : BIT; //Y1.14
        bSameSizeCV_Block2_Valve                   : BIT; //Y1.15
        bSameSizeCV_Block1_Valve                   : BIT; //Y2.0
        bTurntable_Press_Valve                     : BIT; //Y2.1
        bTransmitCV_SameSizeSide_Fwd               : BIT; //Y2.2
        bShipping_FanucRobotPower                  : BIT; //Y2.3
        bTransmitCV_DifferentSide_Fwd              : BIT; //Y2.4
        bTransmitCV_DifferentSide_Rev              : BIT; //Y2.5
        bAllocated_AreaLight                       : BIT; //Y2.6
        bTransmitCV_SameSide_Rev                   : BIT; //Y2.7
        bAllocated_SignalTower_RedLamp             : BIT; //Y2.8
        bAllocated_SignalTower_YellowLamp          : BIT; //Y2.9
        bAllocated_SignalTower_GreenLamp           : BIT; //Y2.10
        bAllocated_SignalTower_BlueLamp            : BIT; //Y2.11
        bAllocated_StartPbLamp                     : BIT; //Y2.12
        bAllocated_StopPbLamp                      : BIT; //Y2.13
        bAllocated_ResetPbLamp                     : BIT; //Y2.14
        bAllocated_Buzzer                          : BIT; //Y2.15

    END_STRUCT
END_TYPE

// ---- Library/10_Machine/19_Device/EL2889/ST_OutputTables.TcDUT
TYPE
    ST_OutputTables :
    STRUCT
        Y4  : uni_IntToBool;
        Y5  : uni_IntToBool;
        Y6  : uni_IntToBool;
        Y7  : uni_IntToBool;
        Y8  : uni_IntToBool;
        Y10 : uni_IntToBool;
        Y11 : uni_IntToBool;
        Y0  : uni_IntToBool;
        Y1  : uni_IntToBool;
        Y2  : uni_IntToBool;
    END_STRUCT
END_TYPE

// ---- Library/10_Machine/19_Device/EL2889/uni_OutputModule.TcDUT
TYPE
    uni_OutputModule :
    UNION
        stEbusDO : ST_EbusOutputModule;       // Output table defined based on module allocation.
        stDO     : ST_OutputTable;            // Output table defined based on variable names.
        stDIList : ST_OutputTables; // Output table defined based on Mitsubishi PLC convention.
    END_UNION
END_TYPE

// ---- Library/10_Machine/19_Device/FanucRobot/DUTs/E_ClampAction.TcDUT
{attribute 'qualified_only'}
{attribute 'strict'}
TYPE
    E_ClampAction :
    (
        Undefine := 0, // Clamp no action
        PickUp,        // Clamp catch something.
        Place          // Clamp release something.
    );
END_TYPE

// ---- Library/10_Machine/19_Device/FanucRobot/DUTs/E_FanucRobotOpMode.TcDUT
TYPE E_FanucRobotOpMode :
(
	RSR01 := 1,	// Production mode, allow motion command (Warehouse, AbsMove...etc)
	RSR02, // HomeMode, allow robot home command.
	RSR03	// Parameter mode, allow read/write offset data.
);
END_TYPE

// ---- Library/10_Machine/19_Device/FanucRobot/DUTs/E_PullOutConveyorPosition.TcDUT
{attribute 'qualified_only'}
TYPE
    E_PullOutConveyorPosition :
    (
        Undefined := 0,
        I3_Slide, // The left side when facing the machine’s operating side.
        I4_Slide  // The right side when facing the machine’s operating side.
    );
END_TYPE

// ---- Library/10_Machine/19_Device/FanucRobot/DUTs/E_RobotAddress.TcDUT
{attribute 'qualified_only'}
TYPE E_RobotAddress :
(
	Undefined := 0,
	Address01,
	Address02,
	Address03,
	Address04,
	Address05,
	Address06
);
END_TYPE

// ---- Library/10_Machine/19_Device/FanucRobot/DUTs/ST_AutoMode_ShippingRobot_MoveAbs.TcDUT
TYPE ST_AutoMode_ShippingRobot_MoveAbs :
STRUCT
	Command 	: ST_CommandBasic;
	Status 		: ST_StatusBasic;
	Info 		: ST_RobotRegionMove_Info;
END_STRUCT
END_TYPE

// ---- Library/10_Machine/19_Device/FanucRobot/DUTs/ST_CCD_ZoneUse.TcDUT
TYPE
    ST_CCD_ZoneUse :
    STRUCT
        WareHouseA_ClampA_UseCCD : BIT;
        WareHouseA_ClampB_UseCCD : BIT;
        WareHouseB_ClampA_UseCCD : BIT;
        WareHouseB_ClampB_UseCCD : BIT;
        Bzone_UseCCD             : BIT;
        Czone_UseCCD             : BIT;
        Dzone_UseCCD             : BIT;
        Ezone_UseCCD             : BIT;
        Fzone_UseCCD             : BIT;
        Gzone_UseCCD             : BIT;
        Hzone_UseCCD             : BIT;
        Jzone_UseCCD             : BIT;
        Kzone_UseCCD             : BIT;
    END_STRUCT
END_TYPE

// ---- Library/10_Machine/19_Device/FanucRobot/DUTs/ST_FanucUI1.TcDUT
TYPE ST_FanucUI1 :
    STRUCT
        UI01_IMSP       :BIT; // Always on, False : disable Robot power, stop prog
        UI02_Hold       :BIT; // Always on, False : stop action and stop prog
        UI03_SFSP       :BIT; // Safety speed, false : robot speed reduce to low and safe speed (safety door)
        UI04_CycleStop  :BIT; // True : force stop prog
        UI05_FaultReset :BIT; // F_trig , if servo not power on, then set power on, if power on and got this f_trig, alarm reset
        UI06_Start      :BIT; // True : continue prog who be stop before
        UI07_Home       :BIT; // not useful, fanuc disable this
        UI08_Enable     :BIT; // True : allow robot move
        UI09_RSR1       :BIT; // Select RSR prog1
        UI10_RSR2       :BIT; // Select RSR prog2
        UI11_RSR3       :BIT; // Select RSR prog3
        UI12_RSR4       :BIT; // Select RSR prog4
        UI13_RSR5       :BIT; // Select RSR prog5
        UI14_RSR6       :BIT; // Select RSR prog6
        UI15_RSR7       :BIT; // Select RSR prog7
        UI16_RSR8       :BIT; // Select RSR prog8
        UI17_PNSStrobe  :BIT; // not useful, fanuc disable this
        UI18_ProdStart  :BIT; // not useful, fanuc disable this
        UI19,
        UI20,
        UI21,
        UI22,
        UI23,
        UI24,
        UI25,
        UI26,
        UI27,
        UI28,
        UI29,
        UI30,
        UI31,
        UI32 :BIT;
    END_STRUCT
END_TYPE

// ---- Library/10_Machine/19_Device/FanucRobot/DUTs/ST_FanucUO1.TcDUT
TYPE ST_FanucUO1 :
    STRUCT
        UO01_CmdEnabled  :BIT;
        UO02_SystemReady :BIT;
        UO03_PrgRunning  :BIT;
        UO04_PrgPaused   :BIT;
        UO05_MotionHeld  :BIT;
        UO06_Fault       :BIT;
        UO07_AtPerch     :BIT;
        UO08_TPEnabled   :BIT;
        UO09_BattAlarm   :BIT;
        UO10_Busy        :BIT;
        UO11_ACK1        :BIT;
        UO12_ACK2        :BIT;
        UO13_ACK3        :BIT;
        UO14_ACK4        :BIT;
        UO15_ACK5        :BIT;
        UO16_ACK6        :BIT;
        UO17_ACK7        :BIT;
        UO18_ACK8        :BIT;
        UO19_SNACK       :BIT;
        UO20_Reserved    :BIT;
        UO21,
        UO22,
        UO23,
        UO24,
        UO25,
        UO26,
        UO27,
        UO28,
        UO29,
        UO30,
        UO31,
        UO32 :BIT;
    END_STRUCT
END_TYPE

// ---- Library/10_Machine/19_Device/FanucRobot/DUTs/ST_Fanuc_AbsMove.TcDUT
(* This Struct is for DAS system - Faunc Robot
	handshake for clamp A/B to target position
*)
TYPE ST_Fanuc_AbsMove :
    STRUCT
        nArea1    :BIT; // The 1st bit of the int representing the Area. 
        nArea2    :BIT; // The 2nd bit of the int representing the Area. 
        nArea3    :BIT; // The 3rd bit of the int representing the Area. 
        nArea4    :BIT; // The 4th bit of the int representing the Area. 
        nAddress1 :BIT; // The 1st bit of the int representing the Address. 
        nAddress2 :BIT; // The 2nd bit of the int representing the Address.
        nAddress3 :BIT; // The 3rd bit of the int representing the Address.
        nAddress4 :BIT; // The 4th bit of the int representing the Address.
        nAddress5 :BIT; // The 5th bit of the int representing the Address.
        nAddress6 :BIT; // The 6th bit of the int representing the Address.
        nAddress7 :BIT; // The 7th bit of the int representing the Address.
        bGet      :BIT; // Ture : ClampA goto target to pickup box, False : ClampB goto target to place box
        bReserve1 :BIT; // Spare
        bExecute  :BIT; // True : Send command to Robot to process
        bContinue :BIT; // True : Send command to Robot, that robot do next clamp's job
        bReserve2 :BIT; // Spare
    END_STRUCT
END_TYPE

// ---- Library/10_Machine/19_Device/FanucRobot/DUTs/ST_Fanuc_GeneralCommand.TcDUT
TYPE ST_Fanuc_GeneralCommand :
    STRUCT
        ClampA_Open  :BIT; // Force clampA open
        ClampB_Open  :BIT; // Force clampB open
        Spare3       :BIT; // Spare
        VelocityBit0 :BIT; // Fanuc robot system velocity in % (1~100), bit0
        VelocityBit1 :BIT;
        VelocityBit2 :BIT;
        VelocityBit3 :BIT;
        VelocityBit4 :BIT;
        VelocityBit5 :BIT;
        VelocityBit6 :BIT;
        VelocityBit7 :BIT;
        ClampA_Close :BIT;
        ClampB_Close :BIT;
        Spare14      :BIT;
        SPare15      :BIT;
        Spare16      :BIT;
    END_STRUCT
END_TYPE

// ---- Library/10_Machine/19_Device/FanucRobot/DUTs/ST_Fanuc_GeneralCommand_1.TcDUT
TYPE ST_Fanuc_GeneralCommand_1 :
    STRUCT
        ClampA_Open  :BIT; // Force clampA open
        ClampB_Open  :BIT; // Force clampB open
        Spare3       :BIT; // Spare
        VelocityBit0 :BIT; // Fanuc robot system velocity in % (1~100), bit0
        VelocityBit1 :BIT;
        VelocityBit2 :BIT;
        VelocityBit3 :BIT;
        VelocityBit4 :BIT;
        VelocityBit5 :BIT;
        VelocityBit6 :BIT;
        VelocityBit7 :BIT;
        ClampA_Close :BIT;
        ClampB_Close :BIT;
        Spare14      :BIT;
        SPare15      :BIT;
        Spare16      :BIT;
    END_STRUCT
END_TYPE

// ---- Library/10_Machine/19_Device/FanucRobot/DUTs/ST_Fanuc_Status.TcDUT
(* This Struct is for DAS system - Faunc Robot handshake for clamp A/B to target position
*)
TYPE
    ST_Fanuc_Status :
    STRUCT
        Done : BIT;       // True : Command process completed
        Error : BIT;      // True : Process has an error
        ErrorID_01 : BIT; // The 1st bit of the int representing the ErrorID. 
        ErrorID_02 : BIT; // The 2nd bit of the int representing the ErrorID. 
        ErrorID_03 : BIT; // The 3rd bit of the int representing the ErrorID. 
        ErrorID_04 : BIT; // The 4th bit of the int representing the ErrorID. 
        ErrorID_05 : BIT; // The 5th bit of the int representing the ErrorID. 
        ErrorID_06 : BIT; // The 6th bit of the int representing the ErrorID. 
        ErrorID_07 : BIT; // The 7th bit of the int representing the ErrorID. 
        ErrorID_08 : BIT; // The 8th bit of the int representing the ErrorID. 
        ErrorID_09 : BIT; // The 9th bit of the int representing the ErrorID. 
        ErrorID_10 : BIT; // The 10th bit of the int representing the ErrorID. 
        Reserve1 : BIT;
        Reserve2 : BIT;
        Notification : BIT;  // True : Robot send this flag to notify PLC for waiting continue cmd
        AllowContinue : BIT; // True :
        WarehouseA : BIT;    // True : The program for warehouse A is running.
        WarehouseB : BIT;    //True:The program for warehouse B is running.
        AbsMoveA : BIT;      //True:The program for AbsMove A is running.
        AbsMoveB : BIT;      //True:The program for AbsMove B is running.
        ClampA_Open : BIT;   //True: ClampA open
        ClampB_Open : BIT;   // True:ClampB open
        ClampA_Sensor : BIT; // True: ClampA sensor detact
        ClampB_Sensor : BIT; //True:CLampB sensor detact
//        RSR1_active : BIT; // True : Robot running in the RSR1 prog
//        RSR2_active : BIT; // True : Robot running in the RSR2 prog
//        RSR3_active : BIT; // True : Robot running in the RSR3 prog
//        BzoneInWork : BIT; // True : Robot in B zone now
//        EzoneInWork : BIT; // True : Robot in E zone now
//        JzoneInWork : BIT; // True : Robot in J zone now

    END_STRUCT
END_TYPE

// ---- Library/10_Machine/19_Device/FanucRobot/DUTs/ST_Fanuc_WarehouseHandshake.TcDUT
(* This Struct is for DAS system - Faunc Robot
	 handshake for Clamp A/B to warehouse pick/place box
*)
TYPE ST_Fanuc_WarehouseHandshake :
    STRUCT
        nLayer1           :BIT; // The 1st bit of the int representing the Layer. 
        nLayer2           :BIT; // The 2nd bit of the int representing the Layer. 
        nLayer3           :BIT; // The 3rd bit of the int representing the Layer. 
        nLayer4           :BIT; // The 4th bit of the int representing the Layer. 
        nSlide1           :BIT; // The 1st bit of the int representing the Slide
        nSlide2           :BIT; // The 2nd bit of the int representing the Slide
        nSlide3           :BIT; // The 3rd bit of the int representing the Slide
        nSlide4           :BIT; // The 4th bit of the int representing the Slide
        nSlide5           :BIT; // The 5th bit of the int representing the Slide
        bTargetWareHouseA :BIT; // True : ClampA's Target is Warehouse A
        bTargetWareHouseB :BIT; // True : ClampA's Target is Warehouse B
        bGet              :BIT; // Ture : ClampA goto target to pickup box, False : ClampB goto target to place box
        bReserve1         :BIT; // Spare
        bExecute          :BIT; // True : Send command to Robot to process
        bContinue         :BIT; // True : Send command to Robot, that robot do next clamp's job
        bReserve2         :BIT; // Spare
    END_STRUCT
END_TYPE

// ---- Library/10_Machine/19_Device/FanucRobot/DUTs/ST_IntToBool.TcDUT
TYPE ST_IntToBool :
UNION
	nInt : INT:=1;
	BitList : ST_BoolList;
END_UNION
END_TYPE

// ---- Library/10_Machine/19_Device/FanucRobot/DUTs/ST_ReadWriteParaCmd.TcDUT
TYPE ST_ReadWriteParaCmd :
	STRUCT
		ReadPara_Execute :BIT;
		WritePara_Execute:BIT;
		ByPassClampSensor : BIT; // True : ByPass clampA and CalmpB sensor
		WareHouseA :BIT; // True : select warehouse A
		WarehouseB :BIT; // True : select warehouse B
		ClampA :BIT; // True : read / write offset data for clamp A
		ClampB :BIT; // True : read / write offset data for clamp B
		Bzone_AllowWork :BIT; //Allow robot move into roundbelt==>Must confirm roundBelt is done and block movement
		Ezone_AllowWork :BIT;
		Jzone_AllowWork :BIT;
		RSR1_Retry :BIT;
		Allow_ClampA_Enter :BIT;
		Allow_ClampB_Enter :BIT;
		Spare14 :BIT;
		Spare15 :BIT;
		Spare16 :BIT;
	END_STRUCT
END_TYPE

// ---- Library/10_Machine/19_Device/FanucRobot/DUTs/ST_ReadWriteParaStatus.TcDUT
TYPE
    ST_ReadWriteParaStatus :
    STRUCT
        ReadCompleted  : BIT; // True : Read Offset data completed
        WriteCompleted : BIT; // True : Write Offset data completed
        Simulation     : BIT; // True : Fanuc robot some value to be force set
        AutoMode       : BIT; // True : Fanuc robot in Auto mode
        T1Mode         : BIT; // True : Fanuc robot in T1 mode, Manual mode in low speed.
        T2Mode         : BIT; // True : Fanuc robot in T2 mode, Manual mode in high speed.
        E_Stop         : BIT; // True : Fanuce robot teach pendant's Estop has be press.
        RSR1_Active    : BIT; // True : RSR1 prog is running
        RSR2_Active    : BIT; // True : RSR2 prog is running
        RSR3_Active    : BIT; // True : RSR3 prog is running
        BzoneInWork    : BIT; // True : Robot request to move in to allocate zone
        BzoneWaitAllow : BIT; //EzoneInWork    : BIT;
        JzoneInWork    : BIT;
    END_STRUCT
END_TYPE

// ---- Library/20_MachineUnits/21_StorageArea/210_Cabinet/DUTs/E_CabinetJob.TcDUT
{attribute 'qualified_only'}
{attribute 'strict'}
TYPE E_CabinetJob :
(
	Idle :=0,
	Initial,
	MoveIn,
	MoveOut,
	MovingOut,
	MovingIn,
	Moved,
	Finish,
	Error
);
END_TYPE

// ---- Library/20_MachineUnits/21_StorageArea/210_Cabinet/DUTs/st_LayerStatus.TcDUT
TYPE st_LayerStatus :
STRUCT
	bSlide1		:	BOOL;
	bSlide2		:	BOOL;
	bSlide3		:	BOOL;
	bSlide4		:	BOOL;
	bSlide5		:	BOOL;
	bSlide6		:	BOOL;
	bSlide7		:	BOOL;
	bSlide8		:	BOOL;
	bSlide9		:	BOOL;
	bSlide10	:	BOOL;
	bSlide11	:	BOOL;
	bSlide12	:	BOOL;
	bSlide13	:	BOOL;
	bSlide14	:	BOOL;
	bSlide15	:	BOOL;
	bSlide16	:	BOOL;
	bSlide17	:	BOOL;
	bSlide18	:	BOOL;
	bSlide19	:	BOOL;
	bSlide20	:	BOOL;
END_STRUCT
END_TYPE

// ---- Library/20_MachineUnits/21_StorageArea/210_Cabinet/DUTs/st_WarehouseLayer.TcDUT
TYPE st_WarehouseLayer :
STRUCT
	bForward		:	BOOL;
	bBackward		:	BOOL;
	stStatus		:	st_LayerStatus;
END_STRUCT
END_TYPE

// ---- Library/20_MachineUnits/21_StorageArea/210_Cabinet/DUTs/st_WarehouseList.TcDUT
TYPE st_WarehouseList :
STRUCT
	A_Side_Layer1	:	ST_WarehouseLayer;
	A_Side_Layer2	:	ST_WarehouseLayer;
	A_Side_Layer3	:	ST_WarehouseLayer;
	A_Side_Layer4	:	ST_WarehouseLayer;
	A_Side_Layer5	:	ST_WarehouseLayer;
	A_Side_Layer6	:	ST_WarehouseLayer;
	A_Side_Layer7	:	ST_WarehouseLayer;
	A_Side_Layer8	:	ST_WarehouseLayer;
	A_Side_Layer9	:	ST_WarehouseLayer;
	A_Side_Layer10	:	ST_WarehouseLayer;
	B_Side_Layer1	:	ST_WarehouseLayer;
	B_Side_Layer2	:	ST_WarehouseLayer;
	B_Side_Layer3	:	ST_WarehouseLayer;
	B_Side_Layer4	:	ST_WarehouseLayer;
	B_Side_Layer5	:	ST_WarehouseLayer;
	B_Side_Layer6	:	ST_WarehouseLayer;
	B_Side_Layer7	:	ST_WarehouseLayer;
	B_Side_Layer8	:	ST_WarehouseLayer;
	B_Side_Layer9	:	ST_WarehouseLayer;
	B_Side_Layer10	:	ST_WarehouseLayer;
END_STRUCT
END_TYPE

// ---- Library/20_MachineUnits/21_StorageArea/210_Cabinet/DUTs/U_Bits_To_stStatus.TcDUT
TYPE U_Bits_To_stStatus :
UNION
	Bits   : ARRAY [1..10] OF BOOL;
	Status : st_LayerStatus;
	
END_UNION
END_TYPE

// ---- Library/20_MachineUnits/21_StorageArea/210_Cabinet/DUTs/_st_LayerStatus.TcDUT
TYPE _st_LayerStatus :
STRUCT
	bSlides		:ARRAY[1..20]OF	BOOL;
END_STRUCT
END_TYPE

// ---- Library/20_MachineUnits/21_StorageArea/210_Cabinet/DUTs/_st_WareHouseLayer.TcDUT
TYPE _st_WareHouseLayer :
STRUCT
	bForward		:	BOOL;
	bBackward		:	BOOL;
	stStatus		:	_st_LayerStatus;
END_STRUCT
END_TYPE

// ---- Library/20_MachineUnits/21_StorageArea/210_Cabinet/DUTs/_st_WarehouseList.TcDUT
TYPE _st_WarehouseList :
STRUCT
	//A倉儲10層狀態
	ASide_Layers	:ARRAY[1..10] OF _ST_WarehouseLayer;
	//B倉儲10層狀態
	BSide_Layers	:ARRAY[1..10] OF _ST_WarehouseLayer;
END_STRUCT
END_TYPE

// ---- Library/20_MachineUnits/21_StorageArea/Duts/E_CabinetJob.TcDUT
{attribute 'qualified_only'}
{attribute 'strict'}
TYPE E_CabinetJob :
(
	Idle :=0,
	Initial,
	MoveIn,
	MoveOut,
	MovingOut,
	MovingIn,
	Moved,
	Finish,
	Error
);
END_TYPE

// ---- Library/20_MachineUnits/21_StorageArea/Duts/E_FeedInAction.TcDUT
{attribute 'qualified_only'}
{attribute 'strict'}
TYPE E_FeedInAction :
(
	Undefined := 0,
	ClampA_WareHouseA,
	ClampA_WareHouseB,
	ClampA_PullOutConveyor,
	ClampB_WareHouseA,
	ClampB_WareHouseB,
	ClampB_PullOutConveyor,
	A_PullOut_B_WareHouseA,
	A_PullOut_B_WareHouseB,
	A_PullOut_B_PullOut,
	A_WareHouseA_B_WareHouseA,
	A_WareHouseA_B_WareHouseB,
	A_WareHouseA_B_PullOut,
	A_WareHouseB_B_WareHouseA,
	A_WareHouseB_B_WareHouseB,
	A_WareHouseB_B_PullOut
);
END_TYPE

// ---- Library/20_MachineUnits/21_StorageArea/Duts/E_ReloadRoundBoxAction.TcDUT
{attribute 'qualified_only'}
{attribute 'strict'}
TYPE E_ReloadRoundBoxAction :
(
	Undefined := 0,
	ClampA_WareHouseA,
	ClampA_WareHouseB,
	ClampB_WareHouseA,
	ClampB_WareHouseB,
	A_WareHouseA_B_WareHouseA,
	A_WareHouseA_B_WareHouseB,
	A_WareHouseB_B_WareHouseA,
	A_WareHouseB_B_WareHouseB
);
END_TYPE

// ---- Library/20_MachineUnits/21_StorageArea/Duts/st_RobotAbsMove_Ctrl.TcDUT
TYPE st_RobotAbsMove_Ctrl :
STRUCT
	bExecute			: BOOL;
	bReset				: BOOL;
	bAbort				: BOOL;
	bOccupied			: BOOL;
END_STRUCT
END_TYPE

// ---- Library/20_MachineUnits/21_StorageArea/Duts/st_RobotAbsMove_Status.TcDUT
TYPE st_RobotAbsMove_Status :
STRUCT
	bBusy	: BOOL;
	bDone	: BOOL;
	bError	: BOOL;
	iErrorID : UDINT;
	Status : STRING;
END_STRUCT
END_TYPE

// ---- Library/20_MachineUnits/21_StorageArea/Duts/st_RobotWarehouseMove_Ctrl.TcDUT
TYPE st_RobotWarehouseMove_Ctrl :
STRUCT
	bExecute			: BOOL;
	bReset				: BOOL;
	bAbort				: BOOL;
	bOccupied			: BOOL;
	bContinue_A			: BOOL;
END_STRUCT
END_TYPE

// ---- Library/20_MachineUnits/21_StorageArea/Duts/st_RobotWarehouseMove_Status.TcDUT
TYPE st_RobotWarehouseMove_Status :
STRUCT
	bBusy	: BOOL;
	bDone	: BOOL;
	bError	: BOOL;
	iErrorID : UDINT;
	Status : STRING;
END_STRUCT
END_TYPE

// ---- Library/20_MachineUnits/21_StorageArea/Duts/ST_StorageService.TcDUT
TYPE
    ST_StorageService :
    STRUCT
        // Automode Feedin empty box with robot 
        AutoMode_FeedInEmptyBoxWithRobot : REFERENCE TO
            ST_AutoMode_FeedInEmptyBox; // Automode : Feedin empty box with robot from Warehouse and Pullout convenyor
        // Automode Reload RoundBelt box with robot
        AutoMode_ReloadRoundBeltBoxWithRobot : REFERENCE TO
            ST_AutoMode_ReloadRoundBeltBox; // Automode : Reload RoundBelt box with robot from warehouse

        //AutoMode UpperFeedInConveyor
        AutoMode_UpperFeedInConveyor : REFERENCE TO ST_Auto_UpperFeedInConveyor;
        //AutoMode AddBoxes
        AutoMode_AddBoxes : REFERENCE TO ST_AutoAddsBoxes;

        //AutoModeUse------手臂區域移動_FeedIn conveyor
        AutoMode_RobotRegionMove_FeedInConveyor : REFERENCE TO ST_AutoMode_RobotRegionMove;
        //AutoModeUse------手臂區域移動_AllocatedConveyor
        AutoMode_RobotRegionMove_AllocatedConveyor : REFERENCE TO ST_AutoMode_RobotRegionMove;
        //AutoModeUse------手臂區域移動_Pullout conveyor
        AutoMode_RobotRegionMove_PullOutConveyor : REFERENCE TO ST_AutoMode_RobotRegionMove;
        //AutoModeUse------手臂區域移動_Buffer area
        AutoMode_RobotRegionMove_BufferArea : REFERENCE TO ST_AutoMode_RobotRegionMove;
        //AutoModeUse------手臂區域移動_RoundBelt
        AutoMode_RobotRegionMove_RoundBelt : REFERENCE TO ST_AutoMode_RobotRegionMove;

        // Pullout 
        AutoMode_PullOutConveyor : REFERENCE TO ST_AutoPullOutConveyor; // AutoMode PullOut Conveyor
        //AutoModeUse*-------手臂絕對位置移動
        AutoMode_RobotAbsMove : REFERENCE TO st_AutoSixAxisAbsMoveParameter;
        //        //AutoModeUse*-------手臂倉儲位置移動
        //        AutoMode_RobotWarehouseMove : st_AutoSixAxisWarehouseParameter;

        //AutoModeUse------倉儲馬達搭配手臂移動
        AutoMode_WarehouseMotoWithRobotMove : REFERENCE TO st_AutoSixAxisWarehouseParameter;
    END_STRUCT
END_TYPE

// ---- Library/20_MachineUnits/22_AllocateArea/Duts/Enums/E_RoundBeltControlAccess.TcDUT
{attribute 'qualified_only'}
{attribute 'strict'}
TYPE E_RoundBeltControlAccess :
(
	Host := 0, // Controlled by C#
	Allocating	, //Controlled by Allocating,
	FanucRobot //Controlled by Robot
);
END_TYPE

// ---- Library/20_MachineUnits/22_AllocateArea/Duts/E_Pistons.TcDUT
{attribute 'qualified_only'}
//{attribute 'strict'}
TYPE E_Pistons :
    (
        //Noon             := -1,
        LoadingBoxRegion := 0,
        ReturnRegion     := 1,
        AllocatedRegion  := 2

    )UINT;
END_TYPE

// ---- Library/20_MachineUnits/22_AllocateArea/Duts/ST_AllocateService.TcDUT
TYPE
    ST_AllocateService :
    STRUCT
        AllocateMoveStructure              : REFERENCE TO st_ads_AllocateMoveStructure;
        AllocateCircleMove                 : REFERENCE TO st_AllocateCircleMoveStructure;
        TurnTableMove                      : REFERENCE TO st_ads_OneAxisMoveWithPosition;
        AutoMode_AllocateBatchMode         : REFERENCE TO ST_AllocationJobBatchMode;
        AutoMode_SimpleAllocation_Batch    : REFERENCE TO ST_AllocationJobBatchMode;
        AutoMode_AllocateBatchMode_Reverse : REFERENCE TO ST_AllocationJobBatchMode;
        AutoMode_RareBoxMove               : REFERENCE TO st_AutoMode_ClampingBoxesJob;
        AutoMode_EmptyBoxMove              : REFERENCE TO st_AutoMode_ClampingBoxesJob;
        AutoMode_BoxMoveReverse            : REFERENCE TO st_AutoMode_ClampingBoxesJob;
        AutoMode_SameSizeCVCamera          : REFERENCE TO ST_AutoMode_TransCVCamera;
        AutoMode_DifferentCVCamera         : REFERENCE TO ST_AutoMode_TransCVCamera;
        AllocateRegionHome                 : REFERENCE TO st_RegionHome;
        AutoMode_PullOutConveyor           : REFERENCE TO ST_AutoPullOutConveyor;
		AutoMode_AllocateCircleMove 	   : REFERENCE TO st_AllocateCircleMoveStructure;
		AutoMode_TurnTableMove 			   : REFERENCE TO st_ads_OneAxisMoveWithPosition;
		AllocateRobotNeedlingMove 		   : REFERENCE TO st_AllocateRobotNeedlingMove;
    END_STRUCT
END_TYPE

// ---- Library/20_MachineUnits/22_AllocateArea/Duts/ST_DuoCylinders.TcDUT
TYPE ST_DuoCylinders :
STRUCT
	Cylinder1 : REFERENCE TO FB_Cylinder;
	Cylinder2 : REFERENCE TO FB_Cylinder;

END_STRUCT
END_TYPE

// ---- Library/20_MachineUnits/22_AllocateArea/Duts/st_RoundBeltAutoSingleMove_Status.TcDUT
TYPE st_RoundBeltAutoSingleMove_Status :
STRUCT
	Busy : BOOL;
	Done : BOOL;
	Error : BOOL;
	Aborted :BOOL;
	ErrorID : UDINT;
	uniqueErrorCode : STRING;
END_STRUCT
END_TYPE

// ---- Library/20_MachineUnits/22_AllocateArea/Duts/Uni_DuoCylinders.TcDUT
TYPE Uni_DuoCylinders :
UNION
	Cylinders 	: REFERENCE TO ARRAY[0..1] OF FB_Cylinder;
	stCylinders	 :ST_DuoCylinders;
END_UNION
END_TYPE

// ---- Library/20_MachineUnits/23_ShippingArea/Duts/ST_ShippingService.TcDUT
TYPE
    ST_ShippingService :
    STRUCT
        AutoMode_ShippingRobot_Left          : REFERENCE TO ST_AutoMode_ShippingRobot_MoveAbs;
        AutoMode_ShippingRobot_Right         : REFERENCE TO ST_AutoMode_ShippingRobot_MoveAbs;
        AutoMode_ShippingRobot_TransmitCVEnd : REFERENCE TO ST_AutoMode_ShippingRobot_MoveAbs;
    END_STRUCT
END_TYPE

// ---- Library/99_Utilities/Duts/E_SignalTowerLampMode.TcDUT
{attribute 'qualified_only'}
{attribute 'strict'}
TYPE E_SignalTowerLampMode :
(
	Disable := 0,
	AlwaysOn,
	Flash_05Hz,
	Flash_1Hz,
	Flash_2Hz
)DINT;
END_TYPE

// ---- Library/99_Utilities/Duts/ST_BoolList.TcDUT
TYPE ST_BoolList :
    STRUCT
        Bit0  :BIT;
        Bit1  :BIT;
        Bit2  :BIT;
        Bit3  :BIT;
        Bit4  :BIT;
        Bit5  :BIT;
        Bit6  :BIT;
        Bit7  :BIT;
        Bit8  :BIT;
        Bit9  :BIT;
        Bit10 :BIT;
        Bit11 :BIT;
        Bit12 :BIT;
        Bit13 :BIT;
        Bit14 :BIT;
        Bit15 :BIT;
    END_STRUCT
END_TYPE

// ---- Library/99_Utilities/Duts/ST_SignalTower.TcDUT
TYPE ST_SignalTower :
STRUCT
	Lamp_Green : BOOL;
	Lamp_Yellow : BOOL;
	Lamp_Red	: BOOL;
	Buzz		: BOOL;
END_STRUCT
END_TYPE

// ---- Library/99_Utilities/Duts/uni_IntToBool.TcDUT
TYPE uni_IntToBool :
UNION
	nInt : INT;
	BitList : ST_BoolList;
END_UNION
END_TYPE

// ---- POUs/ModbusRTU/00_BaseFBs/01_FB_ObjectBase/DUTs/E_MethodStatus_Basic.TcDUT
// Declare the basic level that a method typically goes through, based on PLC Open OOP guidelines.
{attribute 'strict'}
TYPE
    E_MethodStatus_Basic :
    (
        STATE_DORMANT := 0, // In dormant state, do nothing and just wait for the start command.
        STATE_EXECUTING, // In executing state, the state will do something that you coded
        STATE_ABORTING, // In aborting state, stop all ongoing commands.
        STATE_DONE, // In done state, waitting the reset command or execute signal off
        STATE_Aborted, // In aborted state, method is frozen wait reset command or execute signal off
        STATE_ERROR, // In error state, method has been stopped and only can be restart by reset command or execute signal off 
        STATE_RESETTING, // In resetting state, the state will revert the status to its initial values and clear any error signals.
        STATE_Holding, // In Hold state, stop current process
        STATE_Held, // In Held state, waiting the unhold command and keep unit stop
        STATE_UnHold // In UnHold state, reset unit to continue
    ) UDINT;
END_TYPE

// ---- POUs/ModbusRTU/00_BaseFBs/01_FB_ObjectBase/DUTs/ST_CmdContent.TcDUT
TYPE ST_CmdContent :
STRUCT
	SysTime				: STRING;
	Source				: STRING;
	Command				: STRING;
END_STRUCT
END_TYPE

// ---- POUs/ModbusRTU/00_BaseFBs/01_FB_ObjectBase/DUTs/ST_MsgContent.TcDUT
TYPE ST_MsgContent :
STRUCT
	SysTime				: STRING;
	Source				: STRING;
	Message				: STRING;
END_STRUCT
END_TYPE

// ---- POUs/ModbusRTU/SerialComTask/DUTs/un_RS485States.TcDUT
TYPE un_RS485States :
UNION
	arrSensorBySingleModule : ARRAY[0..9] OF ARRAY[0..9] OF BOOL;
	arrSensorByController   : ARRAY[0..99] OF BOOL;
	
END_UNION
END_TYPE

// ---- POUs/ModbusRTU/SerialComTask/DUTs/un_RS485States_all.TcDUT
TYPE un_RS485States_all :
UNION
	arrSensorByController   : ARRAY[0..3] OF ARRAY[0..99] OF BOOL;
	arrSensorAll			: ARRAY[0..399] OF BOOL;
END_UNION
END_TYPE

// ---- Library/10_Machine/11_IOData/GVL_EIP.TcGVL
{attribute 'qualified_only'}
VAR_GLOBAL
END_VAR

// ---- Library/10_Machine/11_IOData/GVL_Input.TcGVL
{attribute 'qualified_only'}
VAR_GLOBAL
	uniDI : uni_InputModule;
END_VAR

